  MoveL (T6208) to (121.16, 117.66, 7.9) mm, rotated rx 180 ry 0 rz -180 deg; joints [0, 0, 0, 0, 0, 0]
  Call Extruder 0.15054
  MoveL (T6209) to (117.66, 121.16, 7.9) mm, rotated rx 180 ry 0 rz -180 deg; joints [0, 0, 0, 0, 0, 0]
  Call Extruder 0.03385
  MoveL (T6210) to (116.55, 121.16, 7.9) mm, rotated rx 180 ry 0 rz -180 deg; joints [0, 0, 0, 0, 0, 0]
  Call Extruder 0.54738
  MoveL (T6211) to (103.84, 108.45, 7.9) mm, rotated rx 180 ry 0 rz -180 deg; joints [0, 0, 0, 0, 0, 0]
  Call Extruder 0.03385
  MoveL (T6212) to (103.84, 107.34, 7.9) mm, rotated rx 180 ry 0 rz -180 deg; joints [0, 0, 0, 0, 0, 0]
  Call Extruder 0.15054
  MoveL (T6213) to (107.34, 103.84, 7.9) mm, rotated rx 180 ry 0 rz -180 deg; joints [0, 0, 0, 0, 0, 0]
  Call Extruder 0.10645
  MoveL (T6214) to (103.84, 103.84, 7.9) mm, rotated rx 180 ry 0 rz -180 deg; joints [0, 0, 0, 0, 0, 0]
  Call Extruder 0.7458
  MoveL (T6215) to (121.16, 121.16, 7.9) mm, rotated rx 180 ry 0 rz -180 deg; joints [0, 0, 0, 0, 0, 0]
  Call Extruder 0.07441
  MoveL (T6216) to (118.71, 121.16, 7.9) mm, rotated rx 180 ry 0 rz -180 deg; joints [0, 0, 0, 0, 0, 0]
  Set speed (45.0 mm/s)
  Call Extruder -1.6
  MoveL (T6217) to (118.71, 121.16, 7.9) mm, rotated rx 180 ry 0 rz -180 deg; joints [0, 0, 0, 0, 0, 0]
  Set speed (120.0 mm/s)
  MoveL (T6218) to (118.71, 121.16, 7.9) mm, rotated rx 180 ry 0 rz -180 deg; joints [0, 0, 0, 0, 0, 0]
  Call Extruder -0.38
  MoveL (T6219) to (119.78, 121.16, 7.9) mm, rotated rx 180 ry 0 rz -180 deg; joints [0, 0, 0, 0, 0, 0]
  Set speed (45.0 mm/s)
  Call Extruder -0.02
  MoveL (T6220) to (119.78, 121.16, 7.9) mm, rotated rx 180 ry 0 rz -180 deg; joints [0, 0, 0, 0, 0, 0]
  Set speed (150.0 mm/s)
  MoveL (T6221) to (119.78, 121.16, 9.9) mm, rotated rx 180 ry 0 rz -180 deg; joints [0, 0, 0, 0, 0, 0]
  MoveL (T6222) to (104.34, 103.54, 9.9) mm, rotated rx 180 ry 0 rz -180 deg; joints [0, 0, 0, 0, 0, 0]
  MoveL (T6223) to (104.34, 103.54, 8.1) mm, rotated rx 180 ry 0 rz -180 deg; joints [0, 0, 0, 0, 0, 0]
  Set speed (40.0 mm/s)
  Call Extruder 2.0
  MoveL (T6224) to (104.34, 103.54, 8.1) mm, rotated rx 180 ry 0 rz -180 deg; joints [0, 0, 0, 0, 0, 0]
  Set speed (25.1 mm/s)
  MoveL (T6225) to (104.34, 103.54, 8.1) mm, rotated rx 180 ry 0 rz -180 deg; joints [0, 0, 0, 0, 0, 0]
  Call Extruder 0.13892
  MoveL (T6226) to (108.9, 103.54, 8.1) mm, rotated rx 180 ry 0 rz -180 deg; joints [0, 0, 0, 0, 0, 0]
  Call Extruder 0.05773
  MoveL (T6227) to (108.9, 105.43, 8.1) mm, rotated rx 180 ry 0 rz -180 deg; joints [0, 0, 0, 0, 0, 0]
  Call Extruder 0.18959
  MoveL (T6228) to (115.12, 105.43, 8.1) mm, rotated rx 180 ry 0 rz -180 deg; joints [0, 0, 0, 0, 0, 0]
  Call Extruder 0.05773
  MoveL (T6229) to (115.12, 103.54, 8.1) mm, rotated rx 180 ry 0 rz -180 deg; joints [0, 0, 0, 0, 0, 0]
  Call Extruder 0.19303
  MoveL (T6230) to (121.46, 103.54, 8.1) mm, rotated rx 180 ry 0 rz -180 deg; joints [0, 0, 0, 0, 0, 0]
  Call Extruder 0.20425
  MoveL (T6231) to (121.46, 110.24, 8.1) mm, rotated rx 180 ry 0 rz -180 deg; joints [0, 0, 0, 0, 0, 0]
  Call Extruder 0.05905
  MoveL (T6232) to (119.52, 110.24, 8.1) mm, rotated rx 180 ry 0 rz -180 deg; joints [0, 0, 0, 0, 0, 0]
  Call Extruder 0.11452
  MoveL (T6233) to (119.52, 114, 8.1) mm, rotated rx 180 ry 0 rz -180 deg; joints [0, 0, 0, 0, 0, 0]
  Call Extruder 0.0591
  MoveL (T6234) to (121.46, 114, 8.1) mm, rotated rx 180 ry 0 rz -180 deg; joints [0, 0, 0, 0, 0, 0]
  Call Extruder 0.2272
  MoveL (T6235) to (121.46, 121.46, 8.1) mm, rotated rx 180 ry 0 rz -180 deg; joints [0, 0, 0, 0, 0, 0]
  Call Extruder 0.54596
  MoveL (T6236) to (103.54, 121.46, 8.1) mm, rotated rx 180 ry 0 rz -180 deg; joints [0, 0, 0, 0, 0, 0]
  Call Extruder 0.54596
  MoveL (T6237) to (103.54, 103.54, 8.1) mm, rotated rx 180 ry 0 rz -180 deg; joints [0, 0, 0, 0, 0, 0]
  Call Extruder 0.02254
  MoveL (T6238) to (104.28, 103.54, 8.1) mm, rotated rx 180 ry 0 rz -180 deg; joints [0, 0, 0, 0, 0, 0]
  Set speed (150.0 mm/s)
  MoveL (T6239) to (103.53, 103.13, 8.1) mm, rotated rx 180 ry 0 rz -180 deg; joints [0, 0, 0, 0, 0, 0]
  Set speed (25.1 mm/s)
  MoveL (T6240) to (103.53, 103.13, 8.1) mm, rotated rx 180 ry 0 rz -180 deg; joints [0, 0, 0, 0, 0, 0]
  Call Extruder 0.1759
  MoveL (T6241) to (109.31, 103.13, 8.1) mm, rotated rx 180 ry 0 rz -180 deg; joints [0, 0, 0, 0, 0, 0]
  Call Extruder 0.05773
  MoveL (T6242) to (109.31, 105.03, 8.1) mm, rotated rx 180 ry 0 rz -180 deg; joints [0, 0, 0, 0, 0, 0]
  Call Extruder 0.1648
  MoveL (T6243) to (114.72, 105.03, 8.1) mm, rotated rx 180 ry 0 rz -180 deg; joints [0, 0, 0, 0, 0, 0]
  Call Extruder 0.05773
  MoveL (T6244) to (114.72, 103.13, 8.1) mm, rotated rx 180 ry 0 rz -180 deg; joints [0, 0, 0, 0, 0, 0]
  Call Extruder 0.21783
  MoveL (T6245) to (121.87, 103.13, 8.1) mm, rotated rx 180 ry 0 rz -180 deg; joints [0, 0, 0, 0, 0, 0]
  Call Extruder 0.22906
  MoveL (T6246) to (121.87, 110.65, 8.1) mm, rotated rx 180 ry 0 rz -180 deg; joints [0, 0, 0, 0, 0, 0]
  Call Extruder 0.05906
  MoveL (T6247) to (119.93, 110.65, 8.1) mm, rotated rx 180 ry 0 rz -180 deg; joints [0, 0, 0, 0, 0, 0]
  Call Extruder 0.08971
  MoveL (T6248) to (119.93, 113.59, 8.1) mm, rotated rx 180 ry 0 rz -180 deg; joints [0, 0, 0, 0, 0, 0]
  Call Extruder 0.0591
  MoveL (T6249) to (121.87, 113.6, 8.1) mm, rotated rx 180 ry 0 rz -180 deg; joints [0, 0, 0, 0, 0, 0]
  Call Extruder 0.25199
  MoveL (T6250) to (121.87, 121.87, 8.1) mm, rotated rx 180 ry 0 rz -180 deg; joints [0, 0, 0, 0, 0, 0]
  Call Extruder 0.57077
  MoveL (T6251) to (103.13, 121.87, 8.1) mm, rotated rx 180 ry 0 rz -180 deg; joints [0, 0, 0, 0, 0, 0]
  Call Extruder 0.57077
  MoveL (T6252) to (103.13, 103.13, 8.1) mm, rotated rx 180 ry 0 rz -180 deg; joints [0, 0, 0, 0, 0, 0]
  Call Extruder 0.01036
  MoveL (T6253) to (103.47, 103.13, 8.1) mm, rotated rx 180 ry 0 rz -180 deg; joints [0, 0, 0, 0, 0, 0]
  Set speed (150.0 mm/s)
  MoveL (T6254) to (102.72, 102.81, 8.1) mm, rotated rx 180 ry 0 rz -180 deg; joints [0, 0, 0, 0, 0, 0]
  Set speed (25.0 mm/s)
  MoveL (T6255) to (102.72, 102.81, 8.1) mm, rotated rx 180 ry 0 rz -180 deg; joints [0, 0, 0, 0, 0, 0]
  Call Extruder 0.00259
  MoveL (T6256) to (102.72, 102.72, 8.1) mm, rotated rx 180 ry 0 rz -180 deg; joints [0, 0, 0, 0, 0, 0]
  Call Extruder 0.21288
  MoveL (T6257) to (109.71, 102.72, 8.1) mm, rotated rx 180 ry 0 rz -180 deg; joints [0, 0, 0, 0, 0, 0]
  Call Extruder 0.05773
  MoveL (T6258) to (109.71, 104.62, 8.1) mm, rotated rx 180 ry 0 rz -180 deg; joints [0, 0, 0, 0, 0, 0]
  Call Extruder 0.06775
  MoveL (T6259) to (111.94, 104.62, 8.1) mm, rotated rx 180 ry 0 rz -180 deg; joints [0, 0, 0, 0, 0, 0]
  Call Extruder 0.05773
  MoveL (T6260) to (111.94, 102.72, 8.1) mm, rotated rx 180 ry 0 rz -180 deg; joints [0, 0, 0, 0, 0, 0]
  Call Extruder 0.00738
  MoveL (T6261) to (112.18, 102.72, 8.1) mm, rotated rx 180 ry 0 rz -180 deg; joints [0, 0, 0, 0, 0, 0]
  Call Extruder 0.05773
  MoveL (T6262) to (112.18, 104.62, 8.1) mm, rotated rx 180 ry 0 rz -180 deg; joints [0, 0, 0, 0, 0, 0]
  Call Extruder 0.06494
  MoveL (T6263) to (114.31, 104.62, 8.1) mm, rotated rx 180 ry 0 rz -180 deg; joints [0, 0, 0, 0, 0, 0]
  Call Extruder 0.05773
  MoveL (T6264) to (114.31, 102.72, 8.1) mm, rotated rx 180 ry 0 rz -180 deg; joints [0, 0, 0, 0, 0, 0]
  Call Extruder 0.24262
  MoveL (T6265) to (122.28, 102.72, 8.1) mm, rotated rx 180 ry 0 rz -180 deg; joints [0, 0, 0, 0, 0, 0]
  Call Extruder 0.25387
  MoveL (T6266) to (122.28, 111.06, 8.1) mm, rotated rx 180 ry 0 rz -180 deg; joints [0, 0, 0, 0, 0, 0]
  Call Extruder 0.05906
  MoveL (T6267) to (120.34, 111.06, 8.1) mm, rotated rx 180 ry 0 rz -180 deg; joints [0, 0, 0, 0, 0, 0]
  Call Extruder 0.06491
  MoveL (T6268) to (120.33, 113.19, 8.1) mm, rotated rx 180 ry 0 rz -180 deg; joints [0, 0, 0, 0, 0, 0]
  Call Extruder 0.05909
  MoveL (T6269) to (122.28, 113.19, 8.1) mm, rotated rx 180 ry 0 rz -180 deg; joints [0, 0, 0, 0, 0, 0]
  Call Extruder 0.27679
  MoveL (T6270) to (122.28, 122.28, 8.1) mm, rotated rx 180 ry 0 rz -180 deg; joints [0, 0, 0, 0, 0, 0]
  Call Extruder 0.59557
  MoveL (T6271) to (102.72, 122.28, 8.1) mm, rotated rx 180 ry 0 rz -180 deg; joints [0, 0, 0, 0, 0, 0]
  Call Extruder 0.59115
  MoveL (T6272) to (102.72, 102.87, 8.1) mm, rotated rx 180 ry 0 rz -180 deg; joints [0, 0, 0, 0, 0, 0]
  Set speed (150.0 mm/s)
  MoveL (T6273) to (102.78, 102.75, 8.1) mm, rotated rx 180 ry 0 rz -180 deg; joints [0, 0, 0, 0, 0, 0]
  Set speed (45.0 mm/s)
  Call Extruder -1.6
  MoveL (T6274) to (102.78, 102.75, 8.1) mm, rotated rx 180 ry 0 rz -180 deg; joints [0, 0, 0, 0, 0, 0]
  Set speed (120.0 mm/s)
  MoveL (T6275) to (102.78, 102.75, 8.1) mm, rotated rx 180 ry 0 rz -180 deg; joints [0, 0, 0, 0, 0, 0]
  Call Extruder -0.05166
  MoveL (T6276) to (102.72, 102.72, 8.1) mm, rotated rx 180 ry 0 rz -180 deg; joints [0, 0, 0, 0, 0, 0]
  Call Extruder -0.32834
  MoveL (T6277) to (103.65, 102.72, 8.1) mm, rotated rx 180 ry 0 rz -180 deg; joints [0, 0, 0, 0, 0, 0]
  Set speed (45.0 mm/s)
  Call Extruder -0.02
  MoveL (T6278) to (103.65, 102.72, 8.1) mm, rotated rx 180 ry 0 rz -180 deg; joints [0, 0, 0, 0, 0, 0]
  Set speed (150.0 mm/s)
  MoveL (T6279) to (103.65, 102.72, 10.1) mm, rotated rx 180 ry 0 rz -180 deg; joints [0, 0, 0, 0, 0, 0]
  MoveL (T6280) to (108.78, 104.69, 10.1) mm, rotated rx 180 ry 0 rz -180 deg; joints [0, 0, 0, 0, 0, 0]
  MoveL (T6281) to (108.78, 104.69, 8.1) mm, rotated rx 180 ry 0 rz -180 deg; joints [0, 0, 0, 0, 0, 0]
  Set speed (40.0 mm/s)
  Call Extruder 2.0
  MoveL (T6282) to (108.78, 104.69, 8.1) mm, rotated rx 180 ry 0 rz -180 deg; joints [0, 0, 0, 0, 0, 0]
  Set speed (25.1 mm/s)
  MoveL (T6283) to (108.78, 104.69, 8.1) mm, rotated rx 180 ry 0 rz -180 deg; joints [0, 0, 0, 0, 0, 0]
  Call Extruder 0.01598
  MoveL (T6284) to (108.43, 105.04, 8.1) mm, rotated rx 180 ry 0 rz -180 deg; joints [0, 0, 0, 0, 0, 0]
  Call Extruder 0.01987
  MoveL (T6285) to (108.43, 104.43, 8.1) mm, rotated rx 180 ry 0 rz -180 deg; joints [0, 0, 0, 0, 0, 0]
  Call Extruder 0.01598
  MoveL (T6286) to (108.78, 104.08, 8.1) mm, rotated rx 180 ry 0 rz -180 deg; joints [0, 0, 0, 0, 0, 0]
  Set speed (45.0 mm/s)
  Call Extruder -1.6
  MoveL (T6287) to (108.78, 104.08, 8.1) mm, rotated rx 180 ry 0 rz -180 deg; joints [0, 0, 0, 0, 0, 0]
  Set speed (120.0 mm/s)
  MoveL (T6288) to (108.78, 104.08, 8.1) mm, rotated rx 180 ry 0 rz -180 deg; joints [0, 0, 0, 0, 0, 0]
  Call Extruder -0.17547
  MoveL (T6289) to (108.43, 104.43, 8.1) mm, rotated rx 180 ry 0 rz -180 deg; joints [0, 0, 0, 0, 0, 0]
  Call Extruder -0.20453
  MoveL (T6290) to (108.43, 105, 8.1) mm, rotated rx 180 ry 0 rz -180 deg; joints [0, 0, 0, 0, 0, 0]
  Set speed (45.0 mm/s)
  Call Extruder -0.02
  MoveL (T6291) to (108.43, 105, 8.1) mm, rotated rx 180 ry 0 rz -180 deg; joints [0, 0, 0, 0, 0, 0]
  Set speed (150.0 mm/s)
  MoveL (T6292) to (108.43, 105, 10.1) mm, rotated rx 180 ry 0 rz -180 deg; joints [0, 0, 0, 0, 0, 0]
  MoveL (T6293) to (115.13, 105.79, 10.1) mm, rotated rx 180 ry 0 rz -180 deg; joints [0, 0, 0, 0, 0, 0]
  MoveL (T6294) to (115.13, 105.79, 8.1) mm, rotated rx 180 ry 0 rz -180 deg; joints [0, 0, 0, 0, 0, 0]
  Set speed (40.0 mm/s)
  Call Extruder 2.0
  MoveL (T6295) to (115.13, 105.79, 8.1) mm, rotated rx 180 ry 0 rz -180 deg; joints [0, 0, 0, 0, 0, 0]
  Set speed (25.1 mm/s)
  MoveL (T6296) to (115.13, 105.79, 8.1) mm, rotated rx 180 ry 0 rz -180 deg; joints [0, 0, 0, 0, 0, 0]
  Call Extruder 0.00342
  MoveL (T6297) to (115.21, 105.87, 8.1) mm, rotated rx 180 ry 0 rz -180 deg; joints [0, 0, 0, 0, 0, 0]
  Call Extruder 0.01615
  MoveL (T6298) to (115.74, 105.87, 8.1) mm, rotated rx 180 ry 0 rz -180 deg; joints [0, 0, 0, 0, 0, 0]
  Call Extruder 0.01375
  MoveL (T6299) to (116.06, 105.55, 8.1) mm, rotated rx 180 ry 0 rz -180 deg; joints [0, 0, 0, 0, 0, 0]
  Call Extruder 0.03706
  MoveL (T6300) to (116.06, 104.33, 8.1) mm, rotated rx 180 ry 0 rz -180 deg; joints [0, 0, 0, 0, 0, 0]
  Call Extruder 0.02096
  MoveL (T6301) to (116.55, 103.84, 8.1) mm, rotated rx 180 ry 0 rz -180 deg; joints [0, 0, 0, 0, 0, 0]
  Call Extruder 0.03385
  MoveL (T6302) to (117.66, 103.84, 8.1) mm, rotated rx 180 ry 0 rz -180 deg; joints [0, 0, 0, 0, 0, 0]
  Call Extruder 0.15054
  MoveL (T6303) to (121.16, 107.34, 8.1) mm, rotated rx 180 ry 0 rz -180 deg; joints [0, 0, 0, 0, 0, 0]
  Call Extruder 0.03385
  MoveL (T6304) to (121.16, 108.45, 8.1) mm, rotated rx 180 ry 0 rz -180 deg; joints [0, 0, 0, 0, 0, 0]
  Call Extruder 0.06409
  MoveL (T6305) to (119.67, 109.94, 8.1) mm, rotated rx 180 ry 0 rz -180 deg; joints [0, 0, 0, 0, 0, 0]
  Call Extruder 0.04532
  MoveL (T6306) to (121.16, 109.94, 8.1) mm, rotated rx 180 ry 0 rz -180 deg; joints [0, 0, 0, 0, 0, 0]
  Call Extruder 0.02909
  MoveL (T6307) to (121.16, 108.98, 8.1) mm, rotated rx 180 ry 0 rz -180 deg; joints [0, 0, 0, 0, 0, 0]
  Set speed (45.0 mm/s)
  Call Extruder -1.6
  MoveL (T6308) to (121.16, 108.98, 8.1) mm, rotated rx 180 ry 0 rz -180 deg; joints [0, 0, 0, 0, 0, 0]
  Set speed (120.0 mm/s)
  MoveL (T6309) to (121.16, 108.98, 8.1) mm, rotated rx 180 ry 0 rz -180 deg; joints [0, 0, 0, 0, 0, 0]
  Call Extruder -0.34013
  MoveL (T6310) to (121.16, 109.94, 8.1) mm, rotated rx 180 ry 0 rz -180 deg; joints [0, 0, 0, 0, 0, 0]
  Call Extruder -0.03987
  MoveL (T6311) to (121.04, 109.94, 8.1) mm, rotated rx 180 ry 0 rz -180 deg; joints [0, 0, 0, 0, 0, 0]
  Set speed (45.0 mm/s)
  Call Extruder -0.02
  MoveL (T6312) to (121.04, 109.94, 8.1) mm, rotated rx 180 ry 0 rz -180 deg; joints [0, 0, 0, 0, 0, 0]
  Set speed (150.0 mm/s)
  MoveL (T6313) to (121.04, 109.94, 10.1) mm, rotated rx 180 ry 0 rz -180 deg; joints [0, 0, 0, 0, 0, 0]
  MoveL (T6314) to (118.71, 103.84, 10.1) mm, rotated rx 180 ry 0 rz -180 deg; joints [0, 0, 0, 0, 0, 0]
  MoveL (T6315) to (118.71, 103.84, 8.1) mm, rotated rx 180 ry 0 rz -180 deg; joints [0, 0, 0, 0, 0, 0]
  Set speed (40.0 mm/s)
  Call Extruder 2.0
  MoveL (T6316) to (118.71, 103.84, 8.1) mm, rotated rx 180 ry 0 rz -180 deg; joints [0, 0, 0, 0, 0, 0]
  Set speed (25.1 mm/s)
  MoveL (T6317) to (118.71, 103.84, 8.1) mm, rotated rx 180 ry 0 rz -180 deg; joints [0, 0, 0, 0, 0, 0]
  Call Extruder 0.07441
  MoveL (T6318) to (121.16, 103.84, 8.1) mm, rotated rx 180 ry 0 rz -180 deg; joints [0, 0, 0, 0, 0, 0]
  Call Extruder 0.7458
  MoveL (T6319) to (103.84, 121.16, 8.1) mm, rotated rx 180 ry 0 rz -180 deg; joints [0, 0, 0, 0, 0, 0]
  Call Extruder 0.10645
  MoveL (T6320) to (103.84, 117.66, 8.1) mm, rotated rx 180 ry 0 rz -180 deg; joints [0, 0, 0, 0, 0, 0]
  Call Extruder 0.15054
  MoveL (T6321) to (107.34, 121.16, 8.1) mm, rotated rx 180 ry 0 rz -180 deg; joints [0, 0, 0, 0, 0, 0]
  Call Extruder 0.03385
  MoveL (T6322) to (108.45, 121.16, 8.1) mm, rotated rx 180 ry 0 rz -180 deg; joints [0, 0, 0, 0, 0, 0]
  Call Extruder 0.46387
  MoveL (T6323) to (119.22, 110.39, 8.1) mm, rotated rx 180 ry 0 rz -180 deg; joints [0, 0, 0, 0, 0, 0]
  Call Extruder 0.01165
  MoveL (T6324) to (119.22, 110.01, 8.1) mm, rotated rx 180 ry 0 rz -180 deg; joints [0, 0, 0, 0, 0, 0]
  Call Extruder 0.18382
  MoveL (T6325) to (114.95, 105.74, 8.1) mm, rotated rx 180 ry 0 rz -180 deg; joints [0, 0, 0, 0, 0, 0]
  Call Extruder 0.009
  MoveL (T6326) to (114.66, 105.74, 8.1) mm, rotated rx 180 ry 0 rz -180 deg; joints [0, 0, 0, 0, 0, 0]
  Call Extruder 0.46575
  MoveL (T6327) to (103.84, 116.55, 8.1) mm, rotated rx 180 ry 0 rz -180 deg; joints [0, 0, 0, 0, 0, 0]
  Call Extruder 0.07441
  MoveL (T6328) to (103.84, 114.11, 8.1) mm, rotated rx 180 ry 0 rz -180 deg; joints [0, 0, 0, 0, 0, 0]
  Set speed (45.0 mm/s)
  Call Extruder -1.6
  MoveL (T6329) to (103.84, 114.11, 8.1) mm, rotated rx 180 ry 0 rz -180 deg; joints [0, 0, 0, 0, 0, 0]
  Set speed (120.0 mm/s)
  MoveL (T6330) to (103.84, 114.11, 8.1) mm, rotated rx 180 ry 0 rz -180 deg; joints [0, 0, 0, 0, 0, 0]
  Call Extruder -0.38
  MoveL (T6331) to (103.84, 115.17, 8.1) mm, rotated rx 180 ry 0 rz -180 deg; joints [0, 0, 0, 0, 0, 0]
  Set speed (45.0 mm/s)
  Call Extruder -0.02
  MoveL (T6332) to (103.84, 115.17, 8.1) mm, rotated rx 180 ry 0 rz -180 deg; joints [0, 0, 0, 0, 0, 0]
  Set speed (150.0 mm/s)
  MoveL (T6333) to (103.84, 115.17, 10.1) mm, rotated rx 180 ry 0 rz -180 deg; joints [0, 0, 0, 0, 0, 0]
  MoveL (T6334) to (115.37, 105.64, 10.1) mm, rotated rx 180 ry 0 rz -180 deg; joints [0, 0, 0, 0, 0, 0]
  MoveL (T6335) to (115.37, 105.64, 8.1) mm, rotated rx 180 ry 0 rz -180 deg; joints [0, 0, 0, 0, 0, 0]
  Set speed (40.0 mm/s)
  Call Extruder 2.0
  MoveL (T6336) to (115.37, 105.64, 8.1) mm, rotated rx 180 ry 0 rz -180 deg; joints [0, 0, 0, 0, 0, 0]
  Set speed (25.1 mm/s)
  MoveL (T6337) to (115.37, 105.64, 8.1) mm, rotated rx 180 ry 0 rz -180 deg; joints [0, 0, 0, 0, 0, 0]
  Call Extruder 0.01303
  MoveL (T6338) to (115.66, 105.36, 8.1) mm, rotated rx 180 ry 0 rz -180 deg; joints [0, 0, 0, 0, 0, 0]
  Call Extruder 0.01995
  MoveL (T6339) to (115.66, 104.75, 8.1) mm, rotated rx 180 ry 0 rz -180 deg; joints [0, 0, 0, 0, 0, 0]
  Call Extruder 0.01043
  MoveL (T6340) to (115.43, 104.97, 8.1) mm, rotated rx 180 ry 0 rz -180 deg; joints [0, 0, 0, 0, 0, 0]
  Call Extruder 0.01995
  MoveL (T6341) to (115.43, 104.36, 8.1) mm, rotated rx 180 ry 0 rz -180 deg; joints [0, 0, 0, 0, 0, 0]
  Call Extruder 0.01885
  MoveL (T6342) to (115.84, 103.95, 8.1) mm, rotated rx 180 ry 0 rz -180 deg; joints [0, 0, 0, 0, 0, 0]
  Set speed (45.0 mm/s)
  Call Extruder -1.6
  MoveL (T6343) to (115.84, 103.95, 8.1) mm, rotated rx 180 ry 0 rz -180 deg; joints [0, 0, 0, 0, 0, 0]
  Set speed (120.0 mm/s)
  MoveL (T6344) to (115.84, 103.95, 8.1) mm, rotated rx 180 ry 0 rz -180 deg; joints [0, 0, 0, 0, 0, 0]
  Call Extruder -0.20676
  MoveL (T6345) to (115.43, 104.36, 8.1) mm, rotated rx 180 ry 0 rz -180 deg; joints [0, 0, 0, 0, 0, 0]
  Call Extruder -0.17324
  MoveL (T6346) to (115.43, 104.84, 8.1) mm, rotated rx 180 ry 0 rz -180 deg; joints [0, 0, 0, 0, 0, 0]
  Set speed (45.0 mm/s)
  Call Extruder -0.02
  MoveL (T6347) to (115.43, 104.84, 8.1) mm, rotated rx 180 ry 0 rz -180 deg; joints [0, 0, 0, 0, 0, 0]
  Set speed (150.0 mm/s)
  MoveL (T6348) to (115.43, 104.84, 10.1) mm, rotated rx 180 ry 0 rz -180 deg; joints [0, 0, 0, 0, 0, 0]
  MoveL (T6349) to (121.16, 115.5, 10.1) mm, rotated rx 180 ry 0 rz -180 deg; joints [0, 0, 0, 0, 0, 0]
  MoveL (T6350) to (121.16, 115.5, 8.1) mm, rotated rx 180 ry 0 rz -180 deg; joints [0, 0, 0, 0, 0, 0]
  Set speed (40.0 mm/s)
  Call Extruder 2.0
  MoveL (T6351) to (121.16, 115.5, 8.1) mm, rotated rx 180 ry 0 rz -180 deg; joints [0, 0, 0, 0, 0, 0]
  Set speed (25.1 mm/s)
  MoveL (T6352) to (121.16, 115.5, 8.1) mm, rotated rx 180 ry 0 rz -180 deg; joints [0, 0, 0, 0, 0, 0]
  Call Extruder 0.03627
  MoveL (T6353) to (121.16, 114.31, 8.1) mm, rotated rx 180 ry 0 rz -180 deg; joints [0, 0, 0, 0, 0, 0]
  Call Extruder 0.03814
  MoveL (T6354) to (119.9, 114.31, 8.1) mm, rotated rx 180 ry 0 rz -180 deg; joints [0, 0, 0, 0, 0, 0]
  Call Extruder 0.29503
  MoveL (T6355) to (113.06, 121.16, 8.1) mm, rotated rx 180 ry 0 rz -180 deg; joints [0, 0, 0, 0, 0, 0]
  Call Extruder 0.03385
  MoveL (T6356) to (111.94, 121.16, 8.1) mm, rotated rx 180 ry 0 rz -180 deg; joints [0, 0, 0, 0, 0, 0]
  Call Extruder 0.34896
  MoveL (T6357) to (103.84, 113.06, 8.1) mm, rotated rx 180 ry 0 rz -180 deg; joints [0, 0, 0, 0, 0, 0]
  Call Extruder 0.03385
  MoveL (T6358) to (103.84, 111.94, 8.1) mm, rotated rx 180 ry 0 rz -180 deg; joints [0, 0, 0, 0, 0, 0]
  Call Extruder 0.26733
  MoveL (T6359) to (110.05, 105.74, 8.1) mm, rotated rx 180 ry 0 rz -180 deg; joints [0, 0, 0, 0, 0, 0]
  Call Extruder 0.009
  MoveL (T6360) to (110.34, 105.74, 8.1) mm, rotated rx 180 ry 0 rz -180 deg; joints [0, 0, 0, 0, 0, 0]
  Call Extruder 0.46575
  MoveL (T6361) to (121.16, 116.55, 8.1) mm, rotated rx 180 ry 0 rz -180 deg; joints [0, 0, 0, 0, 0, 0]
  Call Extruder 0.03385
  MoveL (T6362) to (121.16, 117.66, 8.1) mm, rotated rx 180 ry 0 rz -180 deg; joints [0, 0, 0, 0, 0, 0]
  Call Extruder 0.15054
  MoveL (T6363) to (117.66, 121.16, 8.1) mm, rotated rx 180 ry 0 rz -180 deg; joints [0, 0, 0, 0, 0, 0]
  Call Extruder 0.03385
  MoveL (T6364) to (116.55, 121.16, 8.1) mm, rotated rx 180 ry 0 rz -180 deg; joints [0, 0, 0, 0, 0, 0]
  Call Extruder 0.54738
  MoveL (T6365) to (103.84, 108.45, 8.1) mm, rotated rx 180 ry 0 rz -180 deg; joints [0, 0, 0, 0, 0, 0]
  Call Extruder 0.03385
  MoveL (T6366) to (103.84, 107.34, 8.1) mm, rotated rx 180 ry 0 rz -180 deg; joints [0, 0, 0, 0, 0, 0]
  Call Extruder 0.15054
  MoveL (T6367) to (107.34, 103.84, 8.1) mm, rotated rx 180 ry 0 rz -180 deg; joints [0, 0, 0, 0, 0, 0]
  Call Extruder 0.10645
  MoveL (T6368) to (103.84, 103.84, 8.1) mm, rotated rx 180 ry 0 rz -180 deg; joints [0, 0, 0, 0, 0, 0]
  Call Extruder 0.7458
  MoveL (T6369) to (121.16, 121.16, 8.1) mm, rotated rx 180 ry 0 rz -180 deg; joints [0, 0, 0, 0, 0, 0]
  Call Extruder 0.07441
  MoveL (T6370) to (118.71, 121.16, 8.1) mm, rotated rx 180 ry 0 rz -180 deg; joints [0, 0, 0, 0, 0, 0]
  Set speed (45.0 mm/s)
  Call Extruder -1.6
  MoveL (T6371) to (118.71, 121.16, 8.1) mm, rotated rx 180 ry 0 rz -180 deg; joints [0, 0, 0, 0, 0, 0]
  Set speed (120.0 mm/s)
  MoveL (T6372) to (118.71, 121.16, 8.1) mm, rotated rx 180 ry 0 rz -180 deg; joints [0, 0, 0, 0, 0, 0]
  Call Extruder -0.38
  MoveL (T6373) to (119.78, 121.16, 8.1) mm, rotated rx 180 ry 0 rz -180 deg; joints [0, 0, 0, 0, 0, 0]
  Set speed (45.0 mm/s)
  Call Extruder -0.02
  MoveL (T6374) to (119.78, 121.16, 8.1) mm, rotated rx 180 ry 0 rz -180 deg; joints [0, 0, 0, 0, 0, 0]
  Set speed (150.0 mm/s)
  MoveL (T6375) to (119.78, 121.16, 10.1) mm, rotated rx 180 ry 0 rz -180 deg; joints [0, 0, 0, 0, 0, 0]
  MoveL (T6376) to (112.06, 102.81, 10.1) mm, rotated rx 180 ry 0 rz -180 deg; joints [0, 0, 0, 0, 0, 0]
  MoveL (T6377) to (112.06, 102.81, 8.3) mm, rotated rx 180 ry 0 rz -180 deg; joints [0, 0, 0, 0, 0, 0]
  Set speed (40.0 mm/s)
  Call Extruder 2.0
  MoveL (T6378) to (112.06, 102.81, 8.3) mm, rotated rx 180 ry 0 rz -180 deg; joints [0, 0, 0, 0, 0, 0]
  Set speed (25.0 mm/s)
  MoveL (T6379) to (112.06, 102.81, 8.3) mm, rotated rx 180 ry 0 rz -180 deg; joints [0, 0, 0, 0, 0, 0]
  Call Extruder 0.00245
  MoveL (T6380) to (112.06, 102.72, 8.3) mm, rotated rx 180 ry 0 rz -180 deg; joints [0, 0, 0, 0, 0, 0]
  Call Extruder 0.05685
  MoveL (T6381) to (112.06, 104.59, 8.3) mm, rotated rx 180 ry 0 rz -180 deg; joints [0, 0, 0, 0, 0, 0]
  Call Extruder 0.05257
  MoveL (T6382) to (112.06, 102.86, 8.3) mm, rotated rx 180 ry 0 rz -180 deg; joints [0, 0, 0, 0, 0, 0]
  Set speed (150.0 mm/s)
  MoveL (T6383) to (112.12, 102.85, 8.3) mm, rotated rx 180 ry 0 rz -180 deg; joints [0, 0, 0, 0, 0, 0]
  Set speed (45.0 mm/s)
  Call Extruder -1.6
  MoveL (T6384) to (112.12, 102.85, 8.3) mm, rotated rx 180 ry 0 rz -180 deg; joints [0, 0, 0, 0, 0, 0]
  Set speed (120.0 mm/s)
  MoveL (T6385) to (112.12, 102.85, 8.3) mm, rotated rx 180 ry 0 rz -180 deg; joints [0, 0, 0, 0, 0, 0]
  Call Extruder -0.05002
  MoveL (T6386) to (112.06, 102.72, 8.3) mm, rotated rx 180 ry 0 rz -180 deg; joints [0, 0, 0, 0, 0, 0]
  Call Extruder -0.32998
  MoveL (T6387) to (112.06, 103.65, 8.3) mm, rotated rx 180 ry 0 rz -180 deg; joints [0, 0, 0, 0, 0, 0]
  Set speed (45.0 mm/s)
  Call Extruder -0.02
  MoveL (T6388) to (112.06, 103.65, 8.3) mm, rotated rx 180 ry 0 rz -180 deg; joints [0, 0, 0, 0, 0, 0]
  Set speed (150.0 mm/s)
  MoveL (T6389) to (112.06, 103.65, 10.3) mm, rotated rx 180 ry 0 rz -180 deg; joints [0, 0, 0, 0, 0, 0]
  MoveL (T6390) to (104.34, 103.54, 10.3) mm, rotated rx 180 ry 0 rz -180 deg; joints [0, 0, 0, 0, 0, 0]
  MoveL (T6391) to (104.34, 103.54, 8.3) mm, rotated rx 180 ry 0 rz -180 deg; joints [0, 0, 0, 0, 0, 0]
  Set speed (40.0 mm/s)
  Call Extruder 2.0
  MoveL (T6392) to (104.34, 103.54, 8.3) mm, rotated rx 180 ry 0 rz -180 deg; joints [0, 0, 0, 0, 0, 0]
  Set speed (25.0 mm/s)
  MoveL (T6393) to (104.34, 103.54, 8.3) mm, rotated rx 180 ry 0 rz -180 deg; joints [0, 0, 0, 0, 0, 0]
  Call Extruder 0.1423
  MoveL (T6394) to (109.01, 103.54, 8.3) mm, rotated rx 180 ry 0 rz -180 deg; joints [0, 0, 0, 0, 0, 0]
  Call Extruder 0.05773
  MoveL (T6395) to (109.01, 105.43, 8.3) mm, rotated rx 180 ry 0 rz -180 deg; joints [0, 0, 0, 0, 0, 0]
  Call Extruder 0.18235
  MoveL (T6396) to (115, 105.43, 8.3) mm, rotated rx 180 ry 0 rz -180 deg; joints [0, 0, 0, 0, 0, 0]
  Call Extruder 0.05773
  MoveL (T6397) to (115, 103.54, 8.3) mm, rotated rx 180 ry 0 rz -180 deg; joints [0, 0, 0, 0, 0, 0]
  Call Extruder 0.19688
  MoveL (T6398) to (121.46, 103.54, 8.3) mm, rotated rx 180 ry 0 rz -180 deg; joints [0, 0, 0, 0, 0, 0]
  Call Extruder 0.20419
  MoveL (T6399) to (121.46, 110.24, 8.3) mm, rotated rx 180 ry 0 rz -180 deg; joints [0, 0, 0, 0, 0, 0]
  Call Extruder 0.05904
  MoveL (T6400) to (119.52, 110.24, 8.3) mm, rotated rx 180 ry 0 rz -180 deg; joints [0, 0, 0, 0, 0, 0]
  Call Extruder 0.11452
  MoveL (T6401) to (119.52, 114, 8.3) mm, rotated rx 180 ry 0 rz -180 deg; joints [0, 0, 0, 0, 0, 0]
  Call Extruder 0.05909
  MoveL (T6402) to (121.46, 114, 8.3) mm, rotated rx 180 ry 0 rz -180 deg; joints [0, 0, 0, 0, 0, 0]
  Call Extruder 0.22726
  MoveL (T6403) to (121.46, 121.46, 8.3) mm, rotated rx 180 ry 0 rz -180 deg; joints [0, 0, 0, 0, 0, 0]
  Call Extruder 0.54596
  MoveL (T6404) to (103.54, 121.46, 8.3) mm, rotated rx 180 ry 0 rz -180 deg; joints [0, 0, 0, 0, 0, 0]
  Call Extruder 0.54596
  MoveL (T6405) to (103.54, 103.54, 8.3) mm, rotated rx 180 ry 0 rz -180 deg; joints [0, 0, 0, 0, 0, 0]
  Call Extruder 0.02254
  MoveL (T6406) to (104.28, 103.54, 8.3) mm, rotated rx 180 ry 0 rz -180 deg; joints [0, 0, 0, 0, 0, 0]
  Set speed (150.0 mm/s)
  MoveL (T6407) to (103.53, 103.13, 8.3) mm, rotated rx 180 ry 0 rz -180 deg; joints [0, 0, 0, 0, 0, 0]
  Set speed (25.0 mm/s)
  MoveL (T6408) to (103.53, 103.13, 8.3) mm, rotated rx 180 ry 0 rz -180 deg; joints [0, 0, 0, 0, 0, 0]
  Call Extruder 0.17928
  MoveL (T6409) to (109.42, 103.13, 8.3) mm, rotated rx 180 ry 0 rz -180 deg; joints [0, 0, 0, 0, 0, 0]
  Call Extruder 0.05773
  MoveL (T6410) to (109.42, 105.03, 8.3) mm, rotated rx 180 ry 0 rz -180 deg; joints [0, 0, 0, 0, 0, 0]
  Call Extruder 0.15756
  MoveL (T6411) to (114.59, 105.03, 8.3) mm, rotated rx 180 ry 0 rz -180 deg; joints [0, 0, 0, 0, 0, 0]
  Call Extruder 0.05773
  MoveL (T6412) to (114.59, 103.13, 8.3) mm, rotated rx 180 ry 0 rz -180 deg; joints [0, 0, 0, 0, 0, 0]
  Call Extruder 0.22168
  MoveL (T6413) to (121.87, 103.13, 8.3) mm, rotated rx 180 ry 0 rz -180 deg; joints [0, 0, 0, 0, 0, 0]
  Call Extruder 0.22899
  MoveL (T6414) to (121.87, 110.65, 8.3) mm, rotated rx 180 ry 0 rz -180 deg; joints [0, 0, 0, 0, 0, 0]
  Call Extruder 0.05905
  MoveL (T6415) to (119.93, 110.65, 8.3) mm, rotated rx 180 ry 0 rz -180 deg; joints [0, 0, 0, 0, 0, 0]
  Call Extruder 0.08971
  MoveL (T6416) to (119.93, 113.59, 8.3) mm, rotated rx 180 ry 0 rz -180 deg; joints [0, 0, 0, 0, 0, 0]
  Call Extruder 0.05909
  MoveL (T6417) to (121.87, 113.59, 8.3) mm, rotated rx 180 ry 0 rz -180 deg; joints [0, 0, 0, 0, 0, 0]
  Call Extruder 0.25206
  MoveL (T6418) to (121.87, 121.87, 8.3) mm, rotated rx 180 ry 0 rz -180 deg; joints [0, 0, 0, 0, 0, 0]
  Call Extruder 0.57077
  MoveL (T6419) to (103.13, 121.87, 8.3) mm, rotated rx 180 ry 0 rz -180 deg; joints [0, 0, 0, 0, 0, 0]
  Call Extruder 0.57077
  MoveL (T6420) to (103.13, 103.13, 8.3) mm, rotated rx 180 ry 0 rz -180 deg; joints [0, 0, 0, 0, 0, 0]
  Call Extruder 0.01036
  MoveL (T6421) to (103.47, 103.13, 8.3) mm, rotated rx 180 ry 0 rz -180 deg; joints [0, 0, 0, 0, 0, 0]
  Set speed (150.0 mm/s)
  MoveL (T6422) to (102.72, 102.81, 8.3) mm, rotated rx 180 ry 0 rz -180 deg; joints [0, 0, 0, 0, 0, 0]
  Set speed (25.0 mm/s)
  MoveL (T6423) to (102.72, 102.81, 8.3) mm, rotated rx 180 ry 0 rz -180 deg; joints [0, 0, 0, 0, 0, 0]
  Call Extruder 0.00259
  MoveL (T6424) to (102.72, 102.72, 8.3) mm, rotated rx 180 ry 0 rz -180 deg; joints [0, 0, 0, 0, 0, 0]
  Call Extruder 0.21626
  MoveL (T6425) to (109.82, 102.72, 8.3) mm, rotated rx 180 ry 0 rz -180 deg; joints [0, 0, 0, 0, 0, 0]
  Call Extruder 0.05773
  MoveL (T6426) to (109.83, 104.62, 8.3) mm, rotated rx 180 ry 0 rz -180 deg; joints [0, 0, 0, 0, 0, 0]
  Call Extruder 0.13277
  MoveL (T6427) to (114.18, 104.62, 8.3) mm, rotated rx 180 ry 0 rz -180 deg; joints [0, 0, 0, 0, 0, 0]
  Call Extruder 0.05773
  MoveL (T6428) to (114.18, 102.72, 8.3) mm, rotated rx 180 ry 0 rz -180 deg; joints [0, 0, 0, 0, 0, 0]
  Call Extruder 0.24647
  MoveL (T6429) to (122.28, 102.72, 8.3) mm, rotated rx 180 ry 0 rz -180 deg; joints [0, 0, 0, 0, 0, 0]
  Call Extruder 0.2538
  MoveL (T6430) to (122.28, 111.06, 8.3) mm, rotated rx 180 ry 0 rz -180 deg; joints [0, 0, 0, 0, 0, 0]
  Call Extruder 0.05905
  MoveL (T6431) to (120.34, 111.06, 8.3) mm, rotated rx 180 ry 0 rz -180 deg; joints [0, 0, 0, 0, 0, 0]
  Call Extruder 0.06491
  MoveL (T6432) to (120.34, 113.19, 8.3) mm, rotated rx 180 ry 0 rz -180 deg; joints [0, 0, 0, 0, 0, 0]
  Call Extruder 0.05908
  MoveL (T6433) to (122.28, 113.19, 8.3) mm, rotated rx 180 ry 0 rz -180 deg; joints [0, 0, 0, 0, 0, 0]
  Call Extruder 0.27686
  MoveL (T6434) to (122.28, 122.28, 8.3) mm, rotated rx 180 ry 0 rz -180 deg; joints [0, 0, 0, 0, 0, 0]
  Call Extruder 0.59557
  MoveL (T6435) to (102.72, 122.28, 8.3) mm, rotated rx 180 ry 0 rz -180 deg; joints [0, 0, 0, 0, 0, 0]
  Call Extruder 0.59115
  MoveL (T6436) to (102.72, 102.87, 8.3) mm, rotated rx 180 ry 0 rz -180 deg; joints [0, 0, 0, 0, 0, 0]
  Set speed (150.0 mm/s)
  MoveL (T6437) to (102.78, 102.75, 8.3) mm, rotated rx 180 ry 0 rz -180 deg; joints [0, 0, 0, 0, 0, 0]
  Set speed (45.0 mm/s)
  Call Extruder -1.6
  MoveL (T6438) to (102.78, 102.75, 8.3) mm, rotated rx 180 ry 0 rz -180 deg; joints [0, 0, 0, 0, 0, 0]
  Set speed (120.0 mm/s)
  MoveL (T6439) to (102.78, 102.75, 8.3) mm, rotated rx 180 ry 0 rz -180 deg; joints [0, 0, 0, 0, 0, 0]
  Call Extruder -0.05166
  MoveL (T6440) to (102.72, 102.72, 8.3) mm, rotated rx 180 ry 0 rz -180 deg; joints [0, 0, 0, 0, 0, 0]
  Call Extruder -0.32834
  MoveL (T6441) to (103.65, 102.72, 8.3) mm, rotated rx 180 ry 0 rz -180 deg; joints [0, 0, 0, 0, 0, 0]
  Set speed (45.0 mm/s)
  Call Extruder -0.02
  MoveL (T6442) to (103.65, 102.72, 8.3) mm, rotated rx 180 ry 0 rz -180 deg; joints [0, 0, 0, 0, 0, 0]
  Set speed (150.0 mm/s)
  MoveL (T6443) to (103.65, 102.72, 10.3) mm, rotated rx 180 ry 0 rz -180 deg; joints [0, 0, 0, 0, 0, 0]
  MoveL (T6444) to (108.36, 103.99, 10.3) mm, rotated rx 180 ry 0 rz -180 deg; joints [0, 0, 0, 0, 0, 0]
  MoveL (T6445) to (108.36, 103.99, 8.3) mm, rotated rx 180 ry 0 rz -180 deg; joints [0, 0, 0, 0, 0, 0]
  Set speed (40.0 mm/s)
  Call Extruder 2.0
  MoveL (T6446) to (108.36, 103.99, 8.3) mm, rotated rx 180 ry 0 rz -180 deg; joints [0, 0, 0, 0, 0, 0]
  Set speed (25.0 mm/s)
  MoveL (T6447) to (108.36, 103.99, 8.3) mm, rotated rx 180 ry 0 rz -180 deg; joints [0, 0, 0, 0, 0, 0]
  Call Extruder 0.01562
  MoveL (T6448) to (108.7, 104.34, 8.3) mm, rotated rx 180 ry 0 rz -180 deg; joints [0, 0, 0, 0, 0, 0]
  Call Extruder 0.01897
  MoveL (T6449) to (108.71, 104.94, 8.3) mm, rotated rx 180 ry 0 rz -180 deg; joints [0, 0, 0, 0, 0, 0]
  Call Extruder 0.00741
  MoveL (T6450) to (108.54, 104.77, 8.3) mm, rotated rx 180 ry 0 rz -180 deg; joints [0, 0, 0, 0, 0, 0]
  Call Extruder 0.01897
  MoveL (T6451) to (108.54, 105.37, 8.3) mm, rotated rx 180 ry 0 rz -180 deg; joints [0, 0, 0, 0, 0, 0]
  Call Extruder 0.01234
  MoveL (T6452) to (108.82, 105.64, 8.3) mm, rotated rx 180 ry 0 rz -180 deg; joints [0, 0, 0, 0, 0, 0]
  Set speed (45.0 mm/s)
  Call Extruder -1.6
  MoveL (T6453) to (108.82, 105.64, 8.3) mm, rotated rx 180 ry 0 rz -180 deg; joints [0, 0, 0, 0, 0, 0]
  Set speed (120.0 mm/s)
  MoveL (T6454) to (108.82, 105.64, 8.3) mm, rotated rx 180 ry 0 rz -180 deg; joints [0, 0, 0, 0, 0, 0]
  Call Extruder -0.13882
  MoveL (T6455) to (108.54, 105.37, 8.3) mm, rotated rx 180 ry 0 rz -180 deg; joints [0, 0, 0, 0, 0, 0]
  Call Extruder -0.21335
  MoveL (T6456) to (108.54, 104.77, 8.3) mm, rotated rx 180 ry 0 rz -180 deg; joints [0, 0, 0, 0, 0, 0]
  Call Extruder -0.02783
  MoveL (T6457) to (108.6, 104.82, 8.3) mm, rotated rx 180 ry 0 rz -180 deg; joints [0, 0, 0, 0, 0, 0]
  Set speed (45.0 mm/s)
  Call Extruder -0.02
  MoveL (T6458) to (108.6, 104.82, 8.3) mm, rotated rx 180 ry 0 rz -180 deg; joints [0, 0, 0, 0, 0, 0]
  Set speed (150.0 mm/s)
  MoveL (T6459) to (108.6, 104.82, 10.3) mm, rotated rx 180 ry 0 rz -180 deg; joints [0, 0, 0, 0, 0, 0]
  MoveL (T6460) to (103.84, 114.11, 10.3) mm, rotated rx 180 ry 0 rz -180 deg; joints [0, 0, 0, 0, 0, 0]
  MoveL (T6461) to (103.84, 114.11, 8.3) mm, rotated rx 180 ry 0 rz -180 deg; joints [0, 0, 0, 0, 0, 0]
  Set speed (40.0 mm/s)
  Call Extruder 2.0
  MoveL (T6462) to (103.84, 114.11, 8.3) mm, rotated rx 180 ry 0 rz -180 deg; joints [0, 0, 0, 0, 0, 0]
  Set speed (25.0 mm/s)
  MoveL (T6463) to (103.84, 114.11, 8.3) mm, rotated rx 180 ry 0 rz -180 deg; joints [0, 0, 0, 0, 0, 0]
  Call Extruder 0.07441
  MoveL (T6464) to (103.84, 116.55, 8.3) mm, rotated rx 180 ry 0 rz -180 deg; joints [0, 0, 0, 0, 0, 0]
  Call Extruder 0.46574
  MoveL (T6465) to (114.66, 105.74, 8.3) mm, rotated rx 180 ry 0 rz -180 deg; joints [0, 0, 0, 0, 0, 0]
  Call Extruder 0.00901
  MoveL (T6466) to (114.95, 105.74, 8.3) mm, rotated rx 180 ry 0 rz -180 deg; joints [0, 0, 0, 0, 0, 0]
  Call Extruder 0.18383
  MoveL (T6467) to (119.22, 110.01, 8.3) mm, rotated rx 180 ry 0 rz -180 deg; joints [0, 0, 0, 0, 0, 0]
  Call Extruder 0.01163
  MoveL (T6468) to (119.22, 110.39, 8.3) mm, rotated rx 180 ry 0 rz -180 deg; joints [0, 0, 0, 0, 0, 0]
  Call Extruder 0.46388
  MoveL (T6469) to (108.45, 121.16, 8.3) mm, rotated rx 180 ry 0 rz -180 deg; joints [0, 0, 0, 0, 0, 0]
  Call Extruder 0.03385
  MoveL (T6470) to (107.34, 121.16, 8.3) mm, rotated rx 180 ry 0 rz -180 deg; joints [0, 0, 0, 0, 0, 0]
  Call Extruder 0.15054
  MoveL (T6471) to (103.84, 117.66, 8.3) mm, rotated rx 180 ry 0 rz -180 deg; joints [0, 0, 0, 0, 0, 0]
  Call Extruder 0.10645
  MoveL (T6472) to (103.84, 121.16, 8.3) mm, rotated rx 180 ry 0 rz -180 deg; joints [0, 0, 0, 0, 0, 0]
  Call Extruder 0.7458
  MoveL (T6473) to (121.16, 103.84, 8.3) mm, rotated rx 180 ry 0 rz -180 deg; joints [0, 0, 0, 0, 0, 0]
  Call Extruder 0.07441
  MoveL (T6474) to (118.71, 103.84, 8.3) mm, rotated rx 180 ry 0 rz -180 deg; joints [0, 0, 0, 0, 0, 0]
  Set speed (45.0 mm/s)
  Call Extruder -1.6
  MoveL (T6475) to (118.71, 103.84, 8.3) mm, rotated rx 180 ry 0 rz -180 deg; joints [0, 0, 0, 0, 0, 0]
  Set speed (120.0 mm/s)
  MoveL (T6476) to (118.71, 103.84, 8.3) mm, rotated rx 180 ry 0 rz -180 deg; joints [0, 0, 0, 0, 0, 0]
  Call Extruder -0.38
  MoveL (T6477) to (119.78, 103.84, 8.3) mm, rotated rx 180 ry 0 rz -180 deg; joints [0, 0, 0, 0, 0, 0]
  Set speed (45.0 mm/s)
  Call Extruder -0.02
  MoveL (T6478) to (119.78, 103.84, 8.3) mm, rotated rx 180 ry 0 rz -180 deg; joints [0, 0, 0, 0, 0, 0]
  Set speed (150.0 mm/s)
  MoveL (T6479) to (119.78, 103.84, 10.3) mm, rotated rx 180 ry 0 rz -180 deg; joints [0, 0, 0, 0, 0, 0]
  MoveL (T6480) to (115.12, 104.04, 10.3) mm, rotated rx 180 ry 0 rz -180 deg; joints [0, 0, 0, 0, 0, 0]
  MoveL (T6481) to (115.12, 104.04, 8.3) mm, rotated rx 180 ry 0 rz -180 deg; joints [0, 0, 0, 0, 0, 0]
  Set speed (40.0 mm/s)
  Call Extruder 2.0
  MoveL (T6482) to (115.12, 104.04, 8.3) mm, rotated rx 180 ry 0 rz -180 deg; joints [0, 0, 0, 0, 0, 0]
  Set speed (25.0 mm/s)
  MoveL (T6483) to (115.12, 104.04, 8.3) mm, rotated rx 180 ry 0 rz -180 deg; joints [0, 0, 0, 0, 0, 0]
  Call Extruder 0.01928
  MoveL (T6484) to (115.53, 104.45, 8.3) mm, rotated rx 180 ry 0 rz -180 deg; joints [0, 0, 0, 0, 0, 0]
  Call Extruder 0.02088
  MoveL (T6485) to (115.53, 105.08, 8.3) mm, rotated rx 180 ry 0 rz -180 deg; joints [0, 0, 0, 0, 0, 0]
  Call Extruder 0.01928
  MoveL (T6486) to (115.12, 104.67, 8.3) mm, rotated rx 180 ry 0 rz -180 deg; joints [0, 0, 0, 0, 0, 0]
  Set speed (150.0 mm/s)
  MoveL (T6487) to (115.1, 105.87, 8.3) mm, rotated rx 180 ry 0 rz -180 deg; joints [0, 0, 0, 0, 0, 0]
  Set speed (25.0 mm/s)
  MoveL (T6488) to (115.1, 105.87, 8.3) mm, rotated rx 180 ry 0 rz -180 deg; joints [0, 0, 0, 0, 0, 0]
  Call Extruder 0.01572
  MoveL (T6489) to (115.62, 105.87, 8.3) mm, rotated rx 180 ry 0 rz -180 deg; joints [0, 0, 0, 0, 0, 0]
  Call Extruder 0.01375
  MoveL (T6490) to (115.94, 105.55, 8.3) mm, rotated rx 180 ry 0 rz -180 deg; joints [0, 0, 0, 0, 0, 0]
  Call Extruder 0.03321
  MoveL (T6491) to (115.94, 104.46, 8.3) mm, rotated rx 180 ry 0 rz -180 deg; joints [0, 0, 0, 0, 0, 0]
  Call Extruder 0.02641
  MoveL (T6492) to (116.55, 103.84, 8.3) mm, rotated rx 180 ry 0 rz -180 deg; joints [0, 0, 0, 0, 0, 0]
  Call Extruder 0.03385
  MoveL (T6493) to (117.66, 103.84, 8.3) mm, rotated rx 180 ry 0 rz -180 deg; joints [0, 0, 0, 0, 0, 0]
  Call Extruder 0.15054
  MoveL (T6494) to (121.16, 107.34, 8.3) mm, rotated rx 180 ry 0 rz -180 deg; joints [0, 0, 0, 0, 0, 0]
  Call Extruder 0.03385
  MoveL (T6495) to (121.16, 108.45, 8.3) mm, rotated rx 180 ry 0 rz -180 deg; joints [0, 0, 0, 0, 0, 0]
  Call Extruder 0.064
  MoveL (T6496) to (119.67, 109.94, 8.3) mm, rotated rx 180 ry 0 rz -180 deg; joints [0, 0, 0, 0, 0, 0]
  Call Extruder 0.04526
  MoveL (T6497) to (121.16, 109.94, 8.3) mm, rotated rx 180 ry 0 rz -180 deg; joints [0, 0, 0, 0, 0, 0]
  Call Extruder 0.02915
  MoveL (T6498) to (121.16, 108.98, 8.3) mm, rotated rx 180 ry 0 rz -180 deg; joints [0, 0, 0, 0, 0, 0]
  Set speed (45.0 mm/s)
  Call Extruder -1.6
  MoveL (T6499) to (121.16, 108.98, 8.3) mm, rotated rx 180 ry 0 rz -180 deg; joints [0, 0, 0, 0, 0, 0]
  Set speed (120.0 mm/s)
  MoveL (T6500) to (121.16, 108.98, 8.3) mm, rotated rx 180 ry 0 rz -180 deg; joints [0, 0, 0, 0, 0, 0]
  Call Extruder -0.3409
  MoveL (T6501) to (121.16, 109.94, 8.3) mm, rotated rx 180 ry 0 rz -180 deg; joints [0, 0, 0, 0, 0, 0]
  Call Extruder -0.0391
  MoveL (T6502) to (121.05, 109.94, 8.3) mm, rotated rx 180 ry 0 rz -180 deg; joints [0, 0, 0, 0, 0, 0]
  Set speed (45.0 mm/s)
  Call Extruder -0.02
  MoveL (T6503) to (121.05, 109.94, 8.3) mm, rotated rx 180 ry 0 rz -180 deg; joints [0, 0, 0, 0, 0, 0]
  Set speed (150.0 mm/s)
  MoveL (T6504) to (121.05, 109.94, 10.3) mm, rotated rx 180 ry 0 rz -180 deg; joints [0, 0, 0, 0, 0, 0]
  MoveL (T6505) to (121.16, 115.5, 10.3) mm, rotated rx 180 ry 0 rz -180 deg; joints [0, 0, 0, 0, 0, 0]
  MoveL (T6506) to (121.16, 115.5, 8.3) mm, rotated rx 180 ry 0 rz -180 deg; joints [0, 0, 0, 0, 0, 0]
  Set speed (40.0 mm/s)
  Call Extruder 2.0
  MoveL (T6507) to (121.16, 115.5, 8.3) mm, rotated rx 180 ry 0 rz -180 deg; joints [0, 0, 0, 0, 0, 0]
  Set speed (25.0 mm/s)
  MoveL (T6508) to (121.16, 115.5, 8.3) mm, rotated rx 180 ry 0 rz -180 deg; joints [0, 0, 0, 0, 0, 0]
  Call Extruder 0.03633
  MoveL (T6509) to (121.16, 114.31, 8.3) mm, rotated rx 180 ry 0 rz -180 deg; joints [0, 0, 0, 0, 0, 0]
  Call Extruder 0.03807
  MoveL (T6510) to (119.91, 114.31, 8.3) mm, rotated rx 180 ry 0 rz -180 deg; joints [0, 0, 0, 0, 0, 0]
  Call Extruder 0.29512
  MoveL (T6511) to (113.06, 121.16, 8.3) mm, rotated rx 180 ry 0 rz -180 deg; joints [0, 0, 0, 0, 0, 0]
  Call Extruder 0.03385
  MoveL (T6512) to (111.94, 121.16, 8.3) mm, rotated rx 180 ry 0 rz -180 deg; joints [0, 0, 0, 0, 0, 0]
  Call Extruder 0.34896
  MoveL (T6513) to (103.84, 113.06, 8.3) mm, rotated rx 180 ry 0 rz -180 deg; joints [0, 0, 0, 0, 0, 0]
  Call Extruder 0.03385
  MoveL (T6514) to (103.84, 111.94, 8.3) mm, rotated rx 180 ry 0 rz -180 deg; joints [0, 0, 0, 0, 0, 0]
  Call Extruder 0.26732
  MoveL (T6515) to (110.05, 105.74, 8.3) mm, rotated rx 180 ry 0 rz -180 deg; joints [0, 0, 0, 0, 0, 0]
  Call Extruder 0.00901
  MoveL (T6516) to (110.34, 105.74, 8.3) mm, rotated rx 180 ry 0 rz -180 deg; joints [0, 0, 0, 0, 0, 0]
  Call Extruder 0.46574
  MoveL (T6517) to (121.16, 116.55, 8.3) mm, rotated rx 180 ry 0 rz -180 deg; joints [0, 0, 0, 0, 0, 0]
  Call Extruder 0.03385
  MoveL (T6518) to (121.16, 117.66, 8.3) mm, rotated rx 180 ry 0 rz -180 deg; joints [0, 0, 0, 0, 0, 0]
  Call Extruder 0.15054
  MoveL (T6519) to (117.66, 121.16, 8.3) mm, rotated rx 180 ry 0 rz -180 deg; joints [0, 0, 0, 0, 0, 0]
  Call Extruder 0.03385
  MoveL (T6520) to (116.55, 121.16, 8.3) mm, rotated rx 180 ry 0 rz -180 deg; joints [0, 0, 0, 0, 0, 0]
  Call Extruder 0.54738
  MoveL (T6521) to (103.84, 108.45, 8.3) mm, rotated rx 180 ry 0 rz -180 deg; joints [0, 0, 0, 0, 0, 0]
  Call Extruder 0.03385
  MoveL (T6522) to (103.84, 107.34, 8.3) mm, rotated rx 180 ry 0 rz -180 deg; joints [0, 0, 0, 0, 0, 0]
  Call Extruder 0.15054
  MoveL (T6523) to (107.34, 103.84, 8.3) mm, rotated rx 180 ry 0 rz -180 deg; joints [0, 0, 0, 0, 0, 0]
  Call Extruder 0.10645
  MoveL (T6524) to (103.84, 103.84, 8.3) mm, rotated rx 180 ry 0 rz -180 deg; joints [0, 0, 0, 0, 0, 0]
  Call Extruder 0.7458
  MoveL (T6525) to (121.16, 121.16, 8.3) mm, rotated rx 180 ry 0 rz -180 deg; joints [0, 0, 0, 0, 0, 0]
  Call Extruder 0.07441
  MoveL (T6526) to (118.71, 121.16, 8.3) mm, rotated rx 180 ry 0 rz -180 deg; joints [0, 0, 0, 0, 0, 0]
  Set speed (45.0 mm/s)
  Call Extruder -1.6
  MoveL (T6527) to (118.71, 121.16, 8.3) mm, rotated rx 180 ry 0 rz -180 deg; joints [0, 0, 0, 0, 0, 0]
  Set speed (120.0 mm/s)
  MoveL (T6528) to (118.71, 121.16, 8.3) mm, rotated rx 180 ry 0 rz -180 deg; joints [0, 0, 0, 0, 0, 0]
  Call Extruder -0.38
  MoveL (T6529) to (119.78, 121.16, 8.3) mm, rotated rx 180 ry 0 rz -180 deg; joints [0, 0, 0, 0, 0, 0]
  Set speed (45.0 mm/s)
  Call Extruder -0.02
  MoveL (T6530) to (119.78, 121.16, 8.3) mm, rotated rx 180 ry 0 rz -180 deg; joints [0, 0, 0, 0, 0, 0]
  Set speed (150.0 mm/s)
  MoveL (T6531) to (119.78, 121.16, 10.3) mm, rotated rx 180 ry 0 rz -180 deg; joints [0, 0, 0, 0, 0, 0]
  MoveL (T6532) to (104.34, 103.54, 10.3) mm, rotated rx 180 ry 0 rz -180 deg; joints [0, 0, 0, 0, 0, 0]
  MoveL (T6533) to (104.34, 103.54, 8.5) mm, rotated rx 180 ry 0 rz -180 deg; joints [0, 0, 0, 0, 0, 0]
  Set speed (40.0 mm/s)
  Call Extruder 2.0
  MoveL (T6534) to (104.34, 103.54, 8.5) mm, rotated rx 180 ry 0 rz -180 deg; joints [0, 0, 0, 0, 0, 0]
  Set speed (24.5 mm/s)
  MoveL (T6535) to (104.34, 103.54, 8.5) mm, rotated rx 180 ry 0 rz -180 deg; joints [0, 0, 0, 0, 0, 0]
  Call Extruder 0.14568
  MoveL (T6536) to (109.12, 103.54, 8.5) mm, rotated rx 180 ry 0 rz -180 deg; joints [0, 0, 0, 0, 0, 0]
  Call Extruder 0.05774
  MoveL (T6537) to (109.12, 105.43, 8.5) mm, rotated rx 180 ry 0 rz -180 deg; joints [0, 0, 0, 0, 0, 0]
  Call Extruder 0.17512
  MoveL (T6538) to (114.87, 105.43, 8.5) mm, rotated rx 180 ry 0 rz -180 deg; joints [0, 0, 0, 0, 0, 0]
  Call Extruder 0.05774
  MoveL (T6539) to (114.87, 103.54, 8.5) mm, rotated rx 180 ry 0 rz -180 deg; joints [0, 0, 0, 0, 0, 0]
  Call Extruder 0.20074
  MoveL (T6540) to (121.46, 103.54, 8.5) mm, rotated rx 180 ry 0 rz -180 deg; joints [0, 0, 0, 0, 0, 0]
  Call Extruder 0.20412
  MoveL (T6541) to (121.46, 110.24, 8.5) mm, rotated rx 180 ry 0 rz -180 deg; joints [0, 0, 0, 0, 0, 0]
  Call Extruder 0.05903
  MoveL (T6542) to (119.52, 110.24, 8.5) mm, rotated rx 180 ry 0 rz -180 deg; joints [0, 0, 0, 0, 0, 0]
  Call Extruder 0.11452
  MoveL (T6543) to (119.52, 114, 8.5) mm, rotated rx 180 ry 0 rz -180 deg; joints [0, 0, 0, 0, 0, 0]
  Call Extruder 0.05908
  MoveL (T6544) to (121.46, 114, 8.5) mm, rotated rx 180 ry 0 rz -180 deg; joints [0, 0, 0, 0, 0, 0]
  Call Extruder 0.22733
  MoveL (T6545) to (121.46, 121.46, 8.5) mm, rotated rx 180 ry 0 rz -180 deg; joints [0, 0, 0, 0, 0, 0]
  Call Extruder 0.54596
  MoveL (T6546) to (103.54, 121.46, 8.5) mm, rotated rx 180 ry 0 rz -180 deg; joints [0, 0, 0, 0, 0, 0]
  Call Extruder 0.54596
  MoveL (T6547) to (103.54, 103.54, 8.5) mm, rotated rx 180 ry 0 rz -180 deg; joints [0, 0, 0, 0, 0, 0]
  Call Extruder 0.02254
  MoveL (T6548) to (104.28, 103.54, 8.5) mm, rotated rx 180 ry 0 rz -180 deg; joints [0, 0, 0, 0, 0, 0]
  Set speed (150.0 mm/s)
  MoveL (T6549) to (103.53, 103.13, 8.5) mm, rotated rx 180 ry 0 rz -180 deg; joints [0, 0, 0, 0, 0, 0]
  Set speed (24.5 mm/s)
  MoveL (T6550) to (103.53, 103.13, 8.5) mm, rotated rx 180 ry 0 rz -180 deg; joints [0, 0, 0, 0, 0, 0]
  Call Extruder 0.18266
  MoveL (T6551) to (109.53, 103.13, 8.5) mm, rotated rx 180 ry 0 rz -180 deg; joints [0, 0, 0, 0, 0, 0]
  Call Extruder 0.05774
  MoveL (T6552) to (109.53, 105.03, 8.5) mm, rotated rx 180 ry 0 rz -180 deg; joints [0, 0, 0, 0, 0, 0]
  Call Extruder 0.15033
  MoveL (T6553) to (114.46, 105.03, 8.5) mm, rotated rx 180 ry 0 rz -180 deg; joints [0, 0, 0, 0, 0, 0]
  Call Extruder 0.05774
  MoveL (T6554) to (114.47, 103.13, 8.5) mm, rotated rx 180 ry 0 rz -180 deg; joints [0, 0, 0, 0, 0, 0]
  Call Extruder 0.22553
  MoveL (T6555) to (121.87, 103.13, 8.5) mm, rotated rx 180 ry 0 rz -180 deg; joints [0, 0, 0, 0, 0, 0]
  Call Extruder 0.22893
  MoveL (T6556) to (121.87, 110.65, 8.5) mm, rotated rx 180 ry 0 rz -180 deg; joints [0, 0, 0, 0, 0, 0]
  Call Extruder 0.05904
  MoveL (T6557) to (119.93, 110.65, 8.5) mm, rotated rx 180 ry 0 rz -180 deg; joints [0, 0, 0, 0, 0, 0]
  Call Extruder 0.08971
  MoveL (T6558) to (119.93, 113.59, 8.5) mm, rotated rx 180 ry 0 rz -180 deg; joints [0, 0, 0, 0, 0, 0]
  Call Extruder 0.05908
  MoveL (T6559) to (121.87, 113.59, 8.5) mm, rotated rx 180 ry 0 rz -180 deg; joints [0, 0, 0, 0, 0, 0]
  Call Extruder 0.25213
  MoveL (T6560) to (121.87, 121.87, 8.5) mm, rotated rx 180 ry 0 rz -180 deg; joints [0, 0, 0, 0, 0, 0]
  Call Extruder 0.57077
  MoveL (T6561) to (103.13, 121.87, 8.5) mm, rotated rx 180 ry 0 rz -180 deg; joints [0, 0, 0, 0, 0, 0]
  Call Extruder 0.57077
  MoveL (T6562) to (103.13, 103.13, 8.5) mm, rotated rx 180 ry 0 rz -180 deg; joints [0, 0, 0, 0, 0, 0]
  Call Extruder 0.01036
  MoveL (T6563) to (103.47, 103.13, 8.5) mm, rotated rx 180 ry 0 rz -180 deg; joints [0, 0, 0, 0, 0, 0]
  Set speed (150.0 mm/s)
  MoveL (T6564) to (102.72, 102.81, 8.5) mm, rotated rx 180 ry 0 rz -180 deg; joints [0, 0, 0, 0, 0, 0]
  Set speed (24.5 mm/s)
  MoveL (T6565) to (102.72, 102.81, 8.5) mm, rotated rx 180 ry 0 rz -180 deg; joints [0, 0, 0, 0, 0, 0]
  Call Extruder 0.00259
  MoveL (T6566) to (102.72, 102.72, 8.5) mm, rotated rx 180 ry 0 rz -180 deg; joints [0, 0, 0, 0, 0, 0]
  Call Extruder 0.21965
  MoveL (T6567) to (109.94, 102.72, 8.5) mm, rotated rx 180 ry 0 rz -180 deg; joints [0, 0, 0, 0, 0, 0]
  Call Extruder 0.05774
  MoveL (T6568) to (109.94, 104.62, 8.5) mm, rotated rx 180 ry 0 rz -180 deg; joints [0, 0, 0, 0, 0, 0]
  Call Extruder 0.12554
  MoveL (T6569) to (114.06, 104.62, 8.5) mm, rotated rx 180 ry 0 rz -180 deg; joints [0, 0, 0, 0, 0, 0]
  Call Extruder 0.05774
  MoveL (T6570) to (114.06, 102.72, 8.5) mm, rotated rx 180 ry 0 rz -180 deg; joints [0, 0, 0, 0, 0, 0]
  Call Extruder 0.25033
  MoveL (T6571) to (122.28, 102.72, 8.5) mm, rotated rx 180 ry 0 rz -180 deg; joints [0, 0, 0, 0, 0, 0]
  Call Extruder 0.25373
  MoveL (T6572) to (122.28, 111.05, 8.5) mm, rotated rx 180 ry 0 rz -180 deg; joints [0, 0, 0, 0, 0, 0]
  Call Extruder 0.05904
  MoveL (T6573) to (120.34, 111.05, 8.5) mm, rotated rx 180 ry 0 rz -180 deg; joints [0, 0, 0, 0, 0, 0]
  Call Extruder 0.06491
  MoveL (T6574) to (120.34, 113.18, 8.5) mm, rotated rx 180 ry 0 rz -180 deg; joints [0, 0, 0, 0, 0, 0]
  Call Extruder 0.05907
  MoveL (T6575) to (122.28, 113.19, 8.5) mm, rotated rx 180 ry 0 rz -180 deg; joints [0, 0, 0, 0, 0, 0]
  Call Extruder 0.27692
  MoveL (T6576) to (122.28, 122.28, 8.5) mm, rotated rx 180 ry 0 rz -180 deg; joints [0, 0, 0, 0, 0, 0]
  Call Extruder 0.59557
  MoveL (T6577) to (102.72, 122.28, 8.5) mm, rotated rx 180 ry 0 rz -180 deg; joints [0, 0, 0, 0, 0, 0]
  Call Extruder 0.59115
  MoveL (T6578) to (102.72, 102.87, 8.5) mm, rotated rx 180 ry 0 rz -180 deg; joints [0, 0, 0, 0, 0, 0]
  Set speed (150.0 mm/s)
  MoveL (T6579) to (102.78, 102.75, 8.5) mm, rotated rx 180 ry 0 rz -180 deg; joints [0, 0, 0, 0, 0, 0]
  Set speed (45.0 mm/s)
  Call Extruder -1.6
  MoveL (T6580) to (102.78, 102.75, 8.5) mm, rotated rx 180 ry 0 rz -180 deg; joints [0, 0, 0, 0, 0, 0]
  Set speed (120.0 mm/s)
  MoveL (T6581) to (102.78, 102.75, 8.5) mm, rotated rx 180 ry 0 rz -180 deg; joints [0, 0, 0, 0, 0, 0]
  Call Extruder -0.05166
  MoveL (T6582) to (102.72, 102.72, 8.5) mm, rotated rx 180 ry 0 rz -180 deg; joints [0, 0, 0, 0, 0, 0]
  Call Extruder -0.32834
  MoveL (T6583) to (103.65, 102.72, 8.5) mm, rotated rx 180 ry 0 rz -180 deg; joints [0, 0, 0, 0, 0, 0]
  Set speed (45.0 mm/s)
  Call Extruder -0.02
  MoveL (T6584) to (103.65, 102.72, 8.5) mm, rotated rx 180 ry 0 rz -180 deg; joints [0, 0, 0, 0, 0, 0]
  Set speed (150.0 mm/s)
  MoveL (T6585) to (103.65, 102.72, 10.5) mm, rotated rx 180 ry 0 rz -180 deg; joints [0, 0, 0, 0, 0, 0]
  MoveL (T6586) to (109, 104.69, 10.5) mm, rotated rx 180 ry 0 rz -180 deg; joints [0, 0, 0, 0, 0, 0]
  MoveL (T6587) to (109, 104.69, 8.5) mm, rotated rx 180 ry 0 rz -180 deg; joints [0, 0, 0, 0, 0, 0]
  Set speed (40.0 mm/s)
  Call Extruder 2.0
  MoveL (T6588) to (109, 104.69, 8.5) mm, rotated rx 180 ry 0 rz -180 deg; joints [0, 0, 0, 0, 0, 0]
  Set speed (24.5 mm/s)
  MoveL (T6589) to (109, 104.69, 8.5) mm, rotated rx 180 ry 0 rz -180 deg; joints [0, 0, 0, 0, 0, 0]
  Call Extruder 0.01598
  MoveL (T6590) to (108.65, 105.04, 8.5) mm, rotated rx 180 ry 0 rz -180 deg; joints [0, 0, 0, 0, 0, 0]
  Call Extruder 0.01988
  MoveL (T6591) to (108.65, 104.43, 8.5) mm, rotated rx 180 ry 0 rz -180 deg; joints [0, 0, 0, 0, 0, 0]
  Call Extruder 0.01598
  MoveL (T6592) to (109, 104.08, 8.5) mm, rotated rx 180 ry 0 rz -180 deg; joints [0, 0, 0, 0, 0, 0]
  Set speed (45.0 mm/s)
  Call Extruder -1.6
  MoveL (T6593) to (109, 104.08, 8.5) mm, rotated rx 180 ry 0 rz -180 deg; joints [0, 0, 0, 0, 0, 0]
  Set speed (120.0 mm/s)
  MoveL (T6594) to (109, 104.08, 8.5) mm, rotated rx 180 ry 0 rz -180 deg; joints [0, 0, 0, 0, 0, 0]
  Call Extruder -0.17547
  MoveL (T6595) to (108.65, 104.43, 8.5) mm, rotated rx 180 ry 0 rz -180 deg; joints [0, 0, 0, 0, 0, 0]
  Call Extruder -0.20453
  MoveL (T6596) to (108.65, 105, 8.5) mm, rotated rx 180 ry 0 rz -180 deg; joints [0, 0, 0, 0, 0, 0]
  Set speed (45.0 mm/s)
  Call Extruder -0.02
  MoveL (T6597) to (108.65, 105, 8.5) mm, rotated rx 180 ry 0 rz -180 deg; joints [0, 0, 0, 0, 0, 0]
  Set speed (150.0 mm/s)
  MoveL (T6598) to (108.65, 105, 10.5) mm, rotated rx 180 ry 0 rz -180 deg; joints [0, 0, 0, 0, 0, 0]
  MoveL (T6599) to (115.12, 105.64, 10.5) mm, rotated rx 180 ry 0 rz -180 deg; joints [0, 0, 0, 0, 0, 0]
  MoveL (T6600) to (115.12, 105.64, 8.5) mm, rotated rx 180 ry 0 rz -180 deg; joints [0, 0, 0, 0, 0, 0]
  Set speed (40.0 mm/s)
  Call Extruder 2.0
  MoveL (T6601) to (115.12, 105.64, 8.5) mm, rotated rx 180 ry 0 rz -180 deg; joints [0, 0, 0, 0, 0, 0]
  Set speed (24.5 mm/s)
  MoveL (T6602) to (115.12, 105.64, 8.5) mm, rotated rx 180 ry 0 rz -180 deg; joints [0, 0, 0, 0, 0, 0]
  Call Extruder 0.01303
  MoveL (T6603) to (115.4, 105.36, 8.5) mm, rotated rx 180 ry 0 rz -180 deg; joints [0, 0, 0, 0, 0, 0]
  Call Extruder 0.01996
  MoveL (T6604) to (115.4, 104.75, 8.5) mm, rotated rx 180 ry 0 rz -180 deg; joints [0, 0, 0, 0, 0, 0]
  Call Extruder 0.01044
  MoveL (T6605) to (115.18, 104.97, 8.5) mm, rotated rx 180 ry 0 rz -180 deg; joints [0, 0, 0, 0, 0, 0]
  Call Extruder 0.01996
  MoveL (T6606) to (115.18, 104.36, 8.5) mm, rotated rx 180 ry 0 rz -180 deg; joints [0, 0, 0, 0, 0, 0]
  Call Extruder 0.01886
  MoveL (T6607) to (115.59, 103.95, 8.5) mm, rotated rx 180 ry 0 rz -180 deg; joints [0, 0, 0, 0, 0, 0]
  Set speed (150.0 mm/s)
  MoveL (T6608) to (115.28, 105.87, 8.5) mm, rotated rx 180 ry 0 rz -180 deg; joints [0, 0, 0, 0, 0, 0]
  Set speed (24.5 mm/s)
  MoveL (T6609) to (115.28, 105.87, 8.5) mm, rotated rx 180 ry 0 rz -180 deg; joints [0, 0, 0, 0, 0, 0]
  Call Extruder 0.00635
  MoveL (T6610) to (115.49, 105.87, 8.5) mm, rotated rx 180 ry 0 rz -180 deg; joints [0, 0, 0, 0, 0, 0]
  Call Extruder 0.01375
  MoveL (T6611) to (115.81, 105.55, 8.5) mm, rotated rx 180 ry 0 rz -180 deg; joints [0, 0, 0, 0, 0, 0]
  Call Extruder 0.02936
  MoveL (T6612) to (115.81, 104.58, 8.5) mm, rotated rx 180 ry 0 rz -180 deg; joints [0, 0, 0, 0, 0, 0]
  Call Extruder 0.03186
  MoveL (T6613) to (116.55, 103.84, 8.5) mm, rotated rx 180 ry 0 rz -180 deg; joints [0, 0, 0, 0, 0, 0]
  Call Extruder 0.03385
  MoveL (T6614) to (117.66, 103.84, 8.5) mm, rotated rx 180 ry 0 rz -180 deg; joints [0, 0, 0, 0, 0, 0]
  Call Extruder 0.15054
  MoveL (T6615) to (121.16, 107.34, 8.5) mm, rotated rx 180 ry 0 rz -180 deg; joints [0, 0, 0, 0, 0, 0]
  Call Extruder 0.03385
  MoveL (T6616) to (121.16, 108.45, 8.5) mm, rotated rx 180 ry 0 rz -180 deg; joints [0, 0, 0, 0, 0, 0]
  Call Extruder 0.06391
  MoveL (T6617) to (119.67, 109.93, 8.5) mm, rotated rx 180 ry 0 rz -180 deg; joints [0, 0, 0, 0, 0, 0]
  Call Extruder 0.04519
  MoveL (T6618) to (121.16, 109.93, 8.5) mm, rotated rx 180 ry 0 rz -180 deg; joints [0, 0, 0, 0, 0, 0]
  Call Extruder 0.02922
  MoveL (T6619) to (121.16, 108.97, 8.5) mm, rotated rx 180 ry 0 rz -180 deg; joints [0, 0, 0, 0, 0, 0]
  Set speed (45.0 mm/s)
  Call Extruder -1.6
  MoveL (T6620) to (121.16, 108.97, 8.5) mm, rotated rx 180 ry 0 rz -180 deg; joints [0, 0, 0, 0, 0, 0]
  Set speed (120.0 mm/s)
  MoveL (T6621) to (121.16, 108.97, 8.5) mm, rotated rx 180 ry 0 rz -180 deg; joints [0, 0, 0, 0, 0, 0]
  Call Extruder -0.34167
  MoveL (T6622) to (121.16, 109.93, 8.5) mm, rotated rx 180 ry 0 rz -180 deg; joints [0, 0, 0, 0, 0, 0]
  Call Extruder -0.03833
  MoveL (T6623) to (121.05, 109.93, 8.5) mm, rotated rx 180 ry 0 rz -180 deg; joints [0, 0, 0, 0, 0, 0]
  Set speed (45.0 mm/s)
  Call Extruder -0.02
  MoveL (T6624) to (121.05, 109.93, 8.5) mm, rotated rx 180 ry 0 rz -180 deg; joints [0, 0, 0, 0, 0, 0]
  Set speed (150.0 mm/s)
  MoveL (T6625) to (121.05, 109.93, 10.5) mm, rotated rx 180 ry 0 rz -180 deg; joints [0, 0, 0, 0, 0, 0]
  MoveL (T6626) to (118.71, 103.84, 10.5) mm, rotated rx 180 ry 0 rz -180 deg; joints [0, 0, 0, 0, 0, 0]
  MoveL (T6627) to (118.71, 103.84, 8.5) mm, rotated rx 180 ry 0 rz -180 deg; joints [0, 0, 0, 0, 0, 0]
  Set speed (40.0 mm/s)
  Call Extruder 2.0
  MoveL (T6628) to (118.71, 103.84, 8.5) mm, rotated rx 180 ry 0 rz -180 deg; joints [0, 0, 0, 0, 0, 0]
  Set speed (24.5 mm/s)
  MoveL (T6629) to (118.71, 103.84, 8.5) mm, rotated rx 180 ry 0 rz -180 deg; joints [0, 0, 0, 0, 0, 0]
  Call Extruder 0.07441
  MoveL (T6630) to (121.16, 103.84, 8.5) mm, rotated rx 180 ry 0 rz -180 deg; joints [0, 0, 0, 0, 0, 0]
  Call Extruder 0.7458
  MoveL (T6631) to (103.84, 121.16, 8.5) mm, rotated rx 180 ry 0 rz -180 deg; joints [0, 0, 0, 0, 0, 0]
  Call Extruder 0.10645
  MoveL (T6632) to (103.84, 117.66, 8.5) mm, rotated rx 180 ry 0 rz -180 deg; joints [0, 0, 0, 0, 0, 0]
  Call Extruder 0.15054
  MoveL (T6633) to (107.34, 121.16, 8.5) mm, rotated rx 180 ry 0 rz -180 deg; joints [0, 0, 0, 0, 0, 0]
  Call Extruder 0.03385
  MoveL (T6634) to (108.45, 121.16, 8.5) mm, rotated rx 180 ry 0 rz -180 deg; joints [0, 0, 0, 0, 0, 0]
  Call Extruder 0.4639
  MoveL (T6635) to (119.22, 110.39, 8.5) mm, rotated rx 180 ry 0 rz -180 deg; joints [0, 0, 0, 0, 0, 0]
  Call Extruder 0.01161
  MoveL (T6636) to (119.22, 110.01, 8.5) mm, rotated rx 180 ry 0 rz -180 deg; joints [0, 0, 0, 0, 0, 0]
  Call Extruder 0.17832
  MoveL (T6637) to (115.08, 105.87, 8.5) mm, rotated rx 180 ry 0 rz -180 deg; joints [0, 0, 0, 0, 0, 0]
  Call Extruder 0.0036
  MoveL (T6638) to (114.96, 105.87, 8.5) mm, rotated rx 180 ry 0 rz -180 deg; joints [0, 0, 0, 0, 0, 0]
  Call Extruder 0.00552
  MoveL (T6639) to (114.83, 105.74, 8.5) mm, rotated rx 180 ry 0 rz -180 deg; joints [0, 0, 0, 0, 0, 0]
  Call Extruder 0.00541
  MoveL (T6640) to (114.66, 105.74, 8.5) mm, rotated rx 180 ry 0 rz -180 deg; joints [0, 0, 0, 0, 0, 0]
  Call Extruder 0.46573
  MoveL (T6641) to (103.84, 116.55, 8.5) mm, rotated rx 180 ry 0 rz -180 deg; joints [0, 0, 0, 0, 0, 0]
  Call Extruder 0.07441
  MoveL (T6642) to (103.84, 114.11, 8.5) mm, rotated rx 180 ry 0 rz -180 deg; joints [0, 0, 0, 0, 0, 0]
  Set speed (45.0 mm/s)
  Call Extruder -1.6
  MoveL (T6643) to (103.84, 114.11, 8.5) mm, rotated rx 180 ry 0 rz -180 deg; joints [0, 0, 0, 0, 0, 0]
  Set speed (120.0 mm/s)
  MoveL (T6644) to (103.84, 114.11, 8.5) mm, rotated rx 180 ry 0 rz -180 deg; joints [0, 0, 0, 0, 0, 0]
  Call Extruder -0.38
  MoveL (T6645) to (103.84, 115.17, 8.5) mm, rotated rx 180 ry 0 rz -180 deg; joints [0, 0, 0, 0, 0, 0]
  Set speed (45.0 mm/s)
  Call Extruder -0.02
  MoveL (T6646) to (103.84, 115.17, 8.5) mm, rotated rx 180 ry 0 rz -180 deg; joints [0, 0, 0, 0, 0, 0]
  Set speed (150.0 mm/s)
  MoveL (T6647) to (103.84, 115.17, 10.5) mm, rotated rx 180 ry 0 rz -180 deg; joints [0, 0, 0, 0, 0, 0]
  MoveL (T6648) to (118.71, 121.16, 10.5) mm, rotated rx 180 ry 0 rz -180 deg; joints [0, 0, 0, 0, 0, 0]
  MoveL (T6649) to (118.71, 121.16, 8.5) mm, rotated rx 180 ry 0 rz -180 deg; joints [0, 0, 0, 0, 0, 0]
  Set speed (40.0 mm/s)
  Call Extruder 2.0
  MoveL (T6650) to (118.71, 121.16, 8.5) mm, rotated rx 180 ry 0 rz -180 deg; joints [0, 0, 0, 0, 0, 0]
  Set speed (24.5 mm/s)
  MoveL (T6651) to (118.71, 121.16, 8.5) mm, rotated rx 180 ry 0 rz -180 deg; joints [0, 0, 0, 0, 0, 0]
  Call Extruder 0.07441
  MoveL (T6652) to (121.16, 121.16, 8.5) mm, rotated rx 180 ry 0 rz -180 deg; joints [0, 0, 0, 0, 0, 0]
  Call Extruder 0.7458
  MoveL (T6653) to (103.84, 103.84, 8.5) mm, rotated rx 180 ry 0 rz -180 deg; joints [0, 0, 0, 0, 0, 0]
  Call Extruder 0.10645
  MoveL (T6654) to (107.34, 103.84, 8.5) mm, rotated rx 180 ry 0 rz -180 deg; joints [0, 0, 0, 0, 0, 0]
  Call Extruder 0.15054
  MoveL (T6655) to (103.84, 107.34, 8.5) mm, rotated rx 180 ry 0 rz -180 deg; joints [0, 0, 0, 0, 0, 0]
  Call Extruder 0.03385
  MoveL (T6656) to (103.84, 108.45, 8.5) mm, rotated rx 180 ry 0 rz -180 deg; joints [0, 0, 0, 0, 0, 0]
  Call Extruder 0.54738
  MoveL (T6657) to (116.55, 121.16, 8.5) mm, rotated rx 180 ry 0 rz -180 deg; joints [0, 0, 0, 0, 0, 0]
  Call Extruder 0.03385
  MoveL (T6658) to (117.66, 121.16, 8.5) mm, rotated rx 180 ry 0 rz -180 deg; joints [0, 0, 0, 0, 0, 0]
  Call Extruder 0.15054
  MoveL (T6659) to (121.16, 117.66, 8.5) mm, rotated rx 180 ry 0 rz -180 deg; joints [0, 0, 0, 0, 0, 0]
  Call Extruder 0.03385
  MoveL (T6660) to (121.16, 116.55, 8.5) mm, rotated rx 180 ry 0 rz -180 deg; joints [0, 0, 0, 0, 0, 0]
  Call Extruder 0.46573
  MoveL (T6661) to (110.34, 105.74, 8.5) mm, rotated rx 180 ry 0 rz -180 deg; joints [0, 0, 0, 0, 0, 0]
  Call Extruder 0.00902
  MoveL (T6662) to (110.05, 105.74, 8.5) mm, rotated rx 180 ry 0 rz -180 deg; joints [0, 0, 0, 0, 0, 0]
  Call Extruder 0.26731
  MoveL (T6663) to (103.84, 111.94, 8.5) mm, rotated rx 180 ry 0 rz -180 deg; joints [0, 0, 0, 0, 0, 0]
  Call Extruder 0.03385
  MoveL (T6664) to (103.84, 113.06, 8.5) mm, rotated rx 180 ry 0 rz -180 deg; joints [0, 0, 0, 0, 0, 0]
  Call Extruder 0.34896
  MoveL (T6665) to (111.94, 121.16, 8.5) mm, rotated rx 180 ry 0 rz -180 deg; joints [0, 0, 0, 0, 0, 0]
  Call Extruder 0.03385
  MoveL (T6666) to (113.06, 121.16, 8.5) mm, rotated rx 180 ry 0 rz -180 deg; joints [0, 0, 0, 0, 0, 0]
  Call Extruder 0.29521
  MoveL (T6667) to (119.91, 114.3, 8.5) mm, rotated rx 180 ry 0 rz -180 deg; joints [0, 0, 0, 0, 0, 0]
  Call Extruder 0.03801
  MoveL (T6668) to (121.16, 114.3, 8.5) mm, rotated rx 180 ry 0 rz -180 deg; joints [0, 0, 0, 0, 0, 0]
  Call Extruder 0.0364
  MoveL (T6669) to (121.16, 115.5, 8.5) mm, rotated rx 180 ry 0 rz -180 deg; joints [0, 0, 0, 0, 0, 0]
  Set speed (45.0 mm/s)
  Call Extruder -1.6
  MoveL (T6670) to (121.16, 115.5, 8.5) mm, rotated rx 180 ry 0 rz -180 deg; joints [0, 0, 0, 0, 0, 0]
  Set speed (120.0 mm/s)
  MoveL (T6671) to (121.16, 115.5, 8.5) mm, rotated rx 180 ry 0 rz -180 deg; joints [0, 0, 0, 0, 0, 0]
  Call Extruder -0.38
  MoveL (T6672) to (121.16, 114.43, 8.5) mm, rotated rx 180 ry 0 rz -180 deg; joints [0, 0, 0, 0, 0, 0]
  Set speed (45.0 mm/s)
  Call Extruder -0.02
  MoveL (T6673) to (121.16, 114.43, 8.5) mm, rotated rx 180 ry 0 rz -180 deg; joints [0, 0, 0, 0, 0, 0]
  Set speed (150.0 mm/s)
  MoveL (T6674) to (121.16, 114.43, 10.5) mm, rotated rx 180 ry 0 rz -180 deg; joints [0, 0, 0, 0, 0, 0]
  MoveL (T6675) to (104.34, 103.54, 10.5) mm, rotated rx 180 ry 0 rz -180 deg; joints [0, 0, 0, 0, 0, 0]
  MoveL (T6676) to (104.34, 103.54, 8.7) mm, rotated rx 180 ry 0 rz -180 deg; joints [0, 0, 0, 0, 0, 0]
  Set speed (40.0 mm/s)
  Call Extruder 2.0
  MoveL (T6677) to (104.34, 103.54, 8.7) mm, rotated rx 180 ry 0 rz -180 deg; joints [0, 0, 0, 0, 0, 0]
  Set speed (24.5 mm/s)
  MoveL (T6678) to (104.34, 103.54, 8.7) mm, rotated rx 180 ry 0 rz -180 deg; joints [0, 0, 0, 0, 0, 0]
  Call Extruder 0.14906
  MoveL (T6679) to (109.23, 103.54, 8.7) mm, rotated rx 180 ry 0 rz -180 deg; joints [0, 0, 0, 0, 0, 0]
  Call Extruder 0.05774
  MoveL (T6680) to (109.23, 105.44, 8.7) mm, rotated rx 180 ry 0 rz -180 deg; joints [0, 0, 0, 0, 0, 0]
  Call Extruder 0.16788
  MoveL (T6681) to (114.74, 105.44, 8.7) mm, rotated rx 180 ry 0 rz -180 deg; joints [0, 0, 0, 0, 0, 0]
  Call Extruder 0.05774
  MoveL (T6682) to (114.75, 103.54, 8.7) mm, rotated rx 180 ry 0 rz -180 deg; joints [0, 0, 0, 0, 0, 0]
  Call Extruder 0.20459
  MoveL (T6683) to (121.46, 103.54, 8.7) mm, rotated rx 180 ry 0 rz -180 deg; joints [0, 0, 0, 0, 0, 0]
  Call Extruder 0.20405
  MoveL (T6684) to (121.46, 110.24, 8.7) mm, rotated rx 180 ry 0 rz -180 deg; joints [0, 0, 0, 0, 0, 0]
  Call Extruder 0.05902
  MoveL (T6685) to (119.52, 110.24, 8.7) mm, rotated rx 180 ry 0 rz -180 deg; joints [0, 0, 0, 0, 0, 0]
  Call Extruder 0.11452
  MoveL (T6686) to (119.52, 114, 8.7) mm, rotated rx 180 ry 0 rz -180 deg; joints [0, 0, 0, 0, 0, 0]
  Call Extruder 0.05907
  MoveL (T6687) to (121.46, 114, 8.7) mm, rotated rx 180 ry 0 rz -180 deg; joints [0, 0, 0, 0, 0, 0]
  Call Extruder 0.22739
  MoveL (T6688) to (121.46, 121.46, 8.7) mm, rotated rx 180 ry 0 rz -180 deg; joints [0, 0, 0, 0, 0, 0]
  Call Extruder 0.54596
  MoveL (T6689) to (103.54, 121.46, 8.7) mm, rotated rx 180 ry 0 rz -180 deg; joints [0, 0, 0, 0, 0, 0]
  Call Extruder 0.54596
  MoveL (T6690) to (103.54, 103.54, 8.7) mm, rotated rx 180 ry 0 rz -180 deg; joints [0, 0, 0, 0, 0, 0]
  Call Extruder 0.02254
  MoveL (T6691) to (104.28, 103.54, 8.7) mm, rotated rx 180 ry 0 rz -180 deg; joints [0, 0, 0, 0, 0, 0]
  Set speed (150.0 mm/s)
  MoveL (T6692) to (103.53, 103.13, 8.7) mm, rotated rx 180 ry 0 rz -180 deg; joints [0, 0, 0, 0, 0, 0]
  Set speed (24.5 mm/s)
  MoveL (T6693) to (103.53, 103.13, 8.7) mm, rotated rx 180 ry 0 rz -180 deg; joints [0, 0, 0, 0, 0, 0]
  Call Extruder 0.18605
  MoveL (T6694) to (109.64, 103.13, 8.7) mm, rotated rx 180 ry 0 rz -180 deg; joints [0, 0, 0, 0, 0, 0]
  Call Extruder 0.05774
  MoveL (T6695) to (109.64, 105.03, 8.7) mm, rotated rx 180 ry 0 rz -180 deg; joints [0, 0, 0, 0, 0, 0]
  Call Extruder 0.14309
  MoveL (T6696) to (114.34, 105.03, 8.7) mm, rotated rx 180 ry 0 rz -180 deg; joints [0, 0, 0, 0, 0, 0]
  Call Extruder 0.05774
  MoveL (T6697) to (114.34, 103.13, 8.7) mm, rotated rx 180 ry 0 rz -180 deg; joints [0, 0, 0, 0, 0, 0]
  Call Extruder 0.22938
  MoveL (T6698) to (121.87, 103.13, 8.7) mm, rotated rx 180 ry 0 rz -180 deg; joints [0, 0, 0, 0, 0, 0]
  Call Extruder 0.22886
  MoveL (T6699) to (121.87, 110.64, 8.7) mm, rotated rx 180 ry 0 rz -180 deg; joints [0, 0, 0, 0, 0, 0]
  Call Extruder 0.05903
  MoveL (T6700) to (119.93, 110.64, 8.7) mm, rotated rx 180 ry 0 rz -180 deg; joints [0, 0, 0, 0, 0, 0]
  Call Extruder 0.08971
  MoveL (T6701) to (119.93, 113.59, 8.7) mm, rotated rx 180 ry 0 rz -180 deg; joints [0, 0, 0, 0, 0, 0]
  Call Extruder 0.05907
  MoveL (T6702) to (121.87, 113.59, 8.7) mm, rotated rx 180 ry 0 rz -180 deg; joints [0, 0, 0, 0, 0, 0]
  Call Extruder 0.25219
  MoveL (T6703) to (121.87, 121.87, 8.7) mm, rotated rx 180 ry 0 rz -180 deg; joints [0, 0, 0, 0, 0, 0]
  Call Extruder 0.57077
  MoveL (T6704) to (103.13, 121.87, 8.7) mm, rotated rx 180 ry 0 rz -180 deg; joints [0, 0, 0, 0, 0, 0]
  Call Extruder 0.57077
  MoveL (T6705) to (103.13, 103.13, 8.7) mm, rotated rx 180 ry 0 rz -180 deg; joints [0, 0, 0, 0, 0, 0]
  Call Extruder 0.01036
  MoveL (T6706) to (103.47, 103.13, 8.7) mm, rotated rx 180 ry 0 rz -180 deg; joints [0, 0, 0, 0, 0, 0]
  Set speed (150.0 mm/s)
  MoveL (T6707) to (102.72, 102.81, 8.7) mm, rotated rx 180 ry 0 rz -180 deg; joints [0, 0, 0, 0, 0, 0]
  Set speed (24.5 mm/s)
  MoveL (T6708) to (102.72, 102.81, 8.7) mm, rotated rx 180 ry 0 rz -180 deg; joints [0, 0, 0, 0, 0, 0]
  Call Extruder 0.00259
  MoveL (T6709) to (102.72, 102.72, 8.7) mm, rotated rx 180 ry 0 rz -180 deg; joints [0, 0, 0, 0, 0, 0]
  Call Extruder 0.22303
  MoveL (T6710) to (110.05, 102.72, 8.7) mm, rotated rx 180 ry 0 rz -180 deg; joints [0, 0, 0, 0, 0, 0]
  Call Extruder 0.05774
  MoveL (T6711) to (110.05, 104.62, 8.7) mm, rotated rx 180 ry 0 rz -180 deg; joints [0, 0, 0, 0, 0, 0]
  Call Extruder 0.1183
  MoveL (T6712) to (113.93, 104.62, 8.7) mm, rotated rx 180 ry 0 rz -180 deg; joints [0, 0, 0, 0, 0, 0]
  Call Extruder 0.05774
  MoveL (T6713) to (113.93, 102.72, 8.7) mm, rotated rx 180 ry 0 rz -180 deg; joints [0, 0, 0, 0, 0, 0]
  Call Extruder 0.25418
  MoveL (T6714) to (122.28, 102.72, 8.7) mm, rotated rx 180 ry 0 rz -180 deg; joints [0, 0, 0, 0, 0, 0]
  Call Extruder 0.25367
  MoveL (T6715) to (122.28, 111.05, 8.7) mm, rotated rx 180 ry 0 rz -180 deg; joints [0, 0, 0, 0, 0, 0]
  Call Extruder 0.05903
  MoveL (T6716) to (120.34, 111.05, 8.7) mm, rotated rx 180 ry 0 rz -180 deg; joints [0, 0, 0, 0, 0, 0]
  Call Extruder 0.06491
  MoveL (T6717) to (120.34, 113.18, 8.7) mm, rotated rx 180 ry 0 rz -180 deg; joints [0, 0, 0, 0, 0, 0]
  Call Extruder 0.05906
  MoveL (T6718) to (122.28, 113.18, 8.7) mm, rotated rx 180 ry 0 rz -180 deg; joints [0, 0, 0, 0, 0, 0]
  Call Extruder 0.27699
  MoveL (T6719) to (122.28, 122.28, 8.7) mm, rotated rx 180 ry 0 rz -180 deg; joints [0, 0, 0, 0, 0, 0]
  Call Extruder 0.59557
  MoveL (T6720) to (102.72, 122.28, 8.7) mm, rotated rx 180 ry 0 rz -180 deg; joints [0, 0, 0, 0, 0, 0]
  Call Extruder 0.59115
  MoveL (T6721) to (102.72, 102.87, 8.7) mm, rotated rx 180 ry 0 rz -180 deg; joints [0, 0, 0, 0, 0, 0]
  Set speed (150.0 mm/s)
  MoveL (T6722) to (102.78, 102.75, 8.7) mm, rotated rx 180 ry 0 rz -180 deg; joints [0, 0, 0, 0, 0, 0]
  Set speed (45.0 mm/s)
  Call Extruder -1.6
  MoveL (T6723) to (102.78, 102.75, 8.7) mm, rotated rx 180 ry 0 rz -180 deg; joints [0, 0, 0, 0, 0, 0]
  Set speed (120.0 mm/s)
  MoveL (T6724) to (102.78, 102.75, 8.7) mm, rotated rx 180 ry 0 rz -180 deg; joints [0, 0, 0, 0, 0, 0]
  Call Extruder -0.05166
  MoveL (T6725) to (102.72, 102.72, 8.7) mm, rotated rx 180 ry 0 rz -180 deg; joints [0, 0, 0, 0, 0, 0]
  Call Extruder -0.32834
  MoveL (T6726) to (103.65, 102.72, 8.7) mm, rotated rx 180 ry 0 rz -180 deg; joints [0, 0, 0, 0, 0, 0]
  Set speed (45.0 mm/s)
  Call Extruder -0.02
  MoveL (T6727) to (103.65, 102.72, 8.7) mm, rotated rx 180 ry 0 rz -180 deg; joints [0, 0, 0, 0, 0, 0]
  Set speed (150.0 mm/s)
  MoveL (T6728) to (103.65, 102.72, 10.7) mm, rotated rx 180 ry 0 rz -180 deg; joints [0, 0, 0, 0, 0, 0]
  MoveL (T6729) to (108.58, 103.99, 10.7) mm, rotated rx 180 ry 0 rz -180 deg; joints [0, 0, 0, 0, 0, 0]
  MoveL (T6730) to (108.58, 103.99, 8.7) mm, rotated rx 180 ry 0 rz -180 deg; joints [0, 0, 0, 0, 0, 0]
  Set speed (40.0 mm/s)
  Call Extruder 2.0
  MoveL (T6731) to (108.58, 103.99, 8.7) mm, rotated rx 180 ry 0 rz -180 deg; joints [0, 0, 0, 0, 0, 0]
  Set speed (24.5 mm/s)
  MoveL (T6732) to (108.58, 103.99, 8.7) mm, rotated rx 180 ry 0 rz -180 deg; joints [0, 0, 0, 0, 0, 0]
  Call Extruder 0.01562
  MoveL (T6733) to (108.93, 104.34, 8.7) mm, rotated rx 180 ry 0 rz -180 deg; joints [0, 0, 0, 0, 0, 0]
  Call Extruder 0.01897
  MoveL (T6734) to (108.93, 104.94, 8.7) mm, rotated rx 180 ry 0 rz -180 deg; joints [0, 0, 0, 0, 0, 0]
  Call Extruder 0.00741
  MoveL (T6735) to (108.76, 104.77, 8.7) mm, rotated rx 180 ry 0 rz -180 deg; joints [0, 0, 0, 0, 0, 0]
  Call Extruder 0.01897
  MoveL (T6736) to (108.76, 105.37, 8.7) mm, rotated rx 180 ry 0 rz -180 deg; joints [0, 0, 0, 0, 0, 0]
  Call Extruder 0.01235
  MoveL (T6737) to (109.04, 105.64, 8.7) mm, rotated rx 180 ry 0 rz -180 deg; joints [0, 0, 0, 0, 0, 0]
  Set speed (45.0 mm/s)
  Call Extruder -1.6
  MoveL (T6738) to (109.04, 105.64, 8.7) mm, rotated rx 180 ry 0 rz -180 deg; joints [0, 0, 0, 0, 0, 0]
  Set speed (120.0 mm/s)
  MoveL (T6739) to (109.04, 105.64, 8.7) mm, rotated rx 180 ry 0 rz -180 deg; joints [0, 0, 0, 0, 0, 0]
  Call Extruder -0.13884
  MoveL (T6740) to (108.76, 105.37, 8.7) mm, rotated rx 180 ry 0 rz -180 deg; joints [0, 0, 0, 0, 0, 0]
  Call Extruder -0.21338
  MoveL (T6741) to (108.76, 104.77, 8.7) mm, rotated rx 180 ry 0 rz -180 deg; joints [0, 0, 0, 0, 0, 0]
  Call Extruder -0.02778
  MoveL (T6742) to (108.82, 104.83, 8.7) mm, rotated rx 180 ry 0 rz -180 deg; joints [0, 0, 0, 0, 0, 0]
  Set speed (45.0 mm/s)
  Call Extruder -0.02
  MoveL (T6743) to (108.82, 104.83, 8.7) mm, rotated rx 180 ry 0 rz -180 deg; joints [0, 0, 0, 0, 0, 0]
  Set speed (150.0 mm/s)
  MoveL (T6744) to (108.82, 104.83, 10.7) mm, rotated rx 180 ry 0 rz -180 deg; joints [0, 0, 0, 0, 0, 0]
  MoveL (T6745) to (115.46, 104.64, 10.7) mm, rotated rx 180 ry 0 rz -180 deg; joints [0, 0, 0, 0, 0, 0]
  MoveL (T6746) to (115.46, 104.64, 8.7) mm, rotated rx 180 ry 0 rz -180 deg; joints [0, 0, 0, 0, 0, 0]
  Set speed (40.0 mm/s)
  Call Extruder 2.0
  MoveL (T6747) to (115.46, 104.64, 8.7) mm, rotated rx 180 ry 0 rz -180 deg; joints [0, 0, 0, 0, 0, 0]
  Set speed (24.5 mm/s)
  MoveL (T6748) to (115.46, 104.64, 8.7) mm, rotated rx 180 ry 0 rz -180 deg; joints [0, 0, 0, 0, 0, 0]
  Call Extruder 0.01928
  MoveL (T6749) to (115.05, 104.22, 8.7) mm, rotated rx 180 ry 0 rz -180 deg; joints [0, 0, 0, 0, 0, 0]
  Call Extruder 0.02089
  MoveL (T6750) to (115.05, 104.85, 8.7) mm, rotated rx 180 ry 0 rz -180 deg; joints [0, 0, 0, 0, 0, 0]
  Call Extruder 0.01928
  MoveL (T6751) to (115.46, 105.26, 8.7) mm, rotated rx 180 ry 0 rz -180 deg; joints [0, 0, 0, 0, 0, 0]
  Set speed (150.0 mm/s)
  MoveL (T6752) to (116.35, 103.84, 8.7) mm, rotated rx 180 ry 0 rz -180 deg; joints [0, 0, 0, 0, 0, 0]
  Set speed (24.5 mm/s)
  MoveL (T6753) to (116.35, 103.84, 8.7) mm, rotated rx 180 ry 0 rz -180 deg; joints [0, 0, 0, 0, 0, 0]
  Call Extruder 0.02017
  MoveL (T6754) to (115.68, 103.84, 8.7) mm, rotated rx 180 ry 0 rz -180 deg; joints [0, 0, 0, 0, 0, 0]
  Call Extruder 0.02638
  MoveL (T6755) to (115.68, 104.71, 8.7) mm, rotated rx 180 ry 0 rz -180 deg; joints [0, 0, 0, 0, 0, 0]
  Call Extruder 0.03731
  MoveL (T6756) to (116.55, 103.84, 8.7) mm, rotated rx 180 ry 0 rz -180 deg; joints [0, 0, 0, 0, 0, 0]
  Call Extruder 0.03385
  MoveL (T6757) to (117.66, 103.84, 8.7) mm, rotated rx 180 ry 0 rz -180 deg; joints [0, 0, 0, 0, 0, 0]
  Call Extruder 0.15054
  MoveL (T6758) to (121.16, 107.34, 8.7) mm, rotated rx 180 ry 0 rz -180 deg; joints [0, 0, 0, 0, 0, 0]
  Call Extruder 0.03385
  MoveL (T6759) to (121.16, 108.45, 8.7) mm, rotated rx 180 ry 0 rz -180 deg; joints [0, 0, 0, 0, 0, 0]
  Call Extruder 0.06381
  MoveL (T6760) to (119.67, 109.93, 8.7) mm, rotated rx 180 ry 0 rz -180 deg; joints [0, 0, 0, 0, 0, 0]
  Call Extruder 0.04512
  MoveL (T6761) to (121.16, 109.93, 8.7) mm, rotated rx 180 ry 0 rz -180 deg; joints [0, 0, 0, 0, 0, 0]
  Call Extruder 0.02928
  MoveL (T6762) to (121.16, 108.97, 8.7) mm, rotated rx 180 ry 0 rz -180 deg; joints [0, 0, 0, 0, 0, 0]
  Set speed (45.0 mm/s)
  Call Extruder -1.6
  MoveL (T6763) to (121.16, 108.97, 8.7) mm, rotated rx 180 ry 0 rz -180 deg; joints [0, 0, 0, 0, 0, 0]
  Set speed (120.0 mm/s)
  MoveL (T6764) to (121.16, 108.97, 8.7) mm, rotated rx 180 ry 0 rz -180 deg; joints [0, 0, 0, 0, 0, 0]
  Call Extruder -0.34245
  MoveL (T6765) to (121.16, 109.93, 8.7) mm, rotated rx 180 ry 0 rz -180 deg; joints [0, 0, 0, 0, 0, 0]
  Call Extruder -0.03755
  MoveL (T6766) to (121.05, 109.93, 8.7) mm, rotated rx 180 ry 0 rz -180 deg; joints [0, 0, 0, 0, 0, 0]
  Set speed (45.0 mm/s)
  Call Extruder -0.02
  MoveL (T6767) to (121.05, 109.93, 8.7) mm, rotated rx 180 ry 0 rz -180 deg; joints [0, 0, 0, 0, 0, 0]
  Set speed (150.0 mm/s)
  MoveL (T6768) to (121.05, 109.93, 10.7) mm, rotated rx 180 ry 0 rz -180 deg; joints [0, 0, 0, 0, 0, 0]
  MoveL (T6769) to (118.71, 103.84, 10.7) mm, rotated rx 180 ry 0 rz -180 deg; joints [0, 0, 0, 0, 0, 0]
  MoveL (T6770) to (118.71, 103.84, 8.7) mm, rotated rx 180 ry 0 rz -180 deg; joints [0, 0, 0, 0, 0, 0]
  Set speed (40.0 mm/s)
  Call Extruder 2.0
  MoveL (T6771) to (118.71, 103.84, 8.7) mm, rotated rx 180 ry 0 rz -180 deg; joints [0, 0, 0, 0, 0, 0]
  Set speed (24.5 mm/s)
  MoveL (T6772) to (118.71, 103.84, 8.7) mm, rotated rx 180 ry 0 rz -180 deg; joints [0, 0, 0, 0, 0, 0]
  Call Extruder 0.07441
  MoveL (T6773) to (121.16, 103.84, 8.7) mm, rotated rx 180 ry 0 rz -180 deg; joints [0, 0, 0, 0, 0, 0]
  Call Extruder 0.7458
  MoveL (T6774) to (103.84, 121.16, 8.7) mm, rotated rx 180 ry 0 rz -180 deg; joints [0, 0, 0, 0, 0, 0]
  Call Extruder 0.10645
  MoveL (T6775) to (103.84, 117.66, 8.7) mm, rotated rx 180 ry 0 rz -180 deg; joints [0, 0, 0, 0, 0, 0]
  Call Extruder 0.15054
  MoveL (T6776) to (107.34, 121.16, 8.7) mm, rotated rx 180 ry 0 rz -180 deg; joints [0, 0, 0, 0, 0, 0]
  Call Extruder 0.03385
  MoveL (T6777) to (108.45, 121.16, 8.7) mm, rotated rx 180 ry 0 rz -180 deg; joints [0, 0, 0, 0, 0, 0]
  Call Extruder 0.46391
  MoveL (T6778) to (119.22, 110.39, 8.7) mm, rotated rx 180 ry 0 rz -180 deg; joints [0, 0, 0, 0, 0, 0]
  Call Extruder 0.01159
  MoveL (T6779) to (119.22, 110.01, 8.7) mm, rotated rx 180 ry 0 rz -180 deg; joints [0, 0, 0, 0, 0, 0]
  Call Extruder 0.17833
  MoveL (T6780) to (115.08, 105.87, 8.7) mm, rotated rx 180 ry 0 rz -180 deg; joints [0, 0, 0, 0, 0, 0]
  Call Extruder 0.00745
  MoveL (T6781) to (114.83, 105.87, 8.7) mm, rotated rx 180 ry 0 rz -180 deg; joints [0, 0, 0, 0, 0, 0]
  Call Extruder 0.00552
  MoveL (T6782) to (114.71, 105.74, 8.7) mm, rotated rx 180 ry 0 rz -180 deg; joints [0, 0, 0, 0, 0, 0]
  Call Extruder 0.00157
  MoveL (T6783) to (114.66, 105.74, 8.7) mm, rotated rx 180 ry 0 rz -180 deg; joints [0, 0, 0, 0, 0, 0]
  Call Extruder 0.46572
  MoveL (T6784) to (103.84, 116.55, 8.7) mm, rotated rx 180 ry 0 rz -180 deg; joints [0, 0, 0, 0, 0, 0]
  Call Extruder 0.07441
  MoveL (T6785) to (103.84, 114.11, 8.7) mm, rotated rx 180 ry 0 rz -180 deg; joints [0, 0, 0, 0, 0, 0]
  Set speed (45.0 mm/s)
  Call Extruder -1.6
  MoveL (T6786) to (103.84, 114.11, 8.7) mm, rotated rx 180 ry 0 rz -180 deg; joints [0, 0, 0, 0, 0, 0]
  Set speed (120.0 mm/s)
  MoveL (T6787) to (103.84, 114.11, 8.7) mm, rotated rx 180 ry 0 rz -180 deg; joints [0, 0, 0, 0, 0, 0]
  Call Extruder -0.38
  MoveL (T6788) to (103.84, 115.17, 8.7) mm, rotated rx 180 ry 0 rz -180 deg; joints [0, 0, 0, 0, 0, 0]
  Set speed (45.0 mm/s)
  Call Extruder -0.02
  MoveL (T6789) to (103.84, 115.17, 8.7) mm, rotated rx 180 ry 0 rz -180 deg; joints [0, 0, 0, 0, 0, 0]
  Set speed (150.0 mm/s)
  MoveL (T6790) to (103.84, 115.17, 10.7) mm, rotated rx 180 ry 0 rz -180 deg; joints [0, 0, 0, 0, 0, 0]
  MoveL (T6791) to (118.71, 121.16, 10.7) mm, rotated rx 180 ry 0 rz -180 deg; joints [0, 0, 0, 0, 0, 0]
  MoveL (T6792) to (118.71, 121.16, 8.7) mm, rotated rx 180 ry 0 rz -180 deg; joints [0, 0, 0, 0, 0, 0]
  Set speed (40.0 mm/s)
  Call Extruder 2.0
  MoveL (T6793) to (118.71, 121.16, 8.7) mm, rotated rx 180 ry 0 rz -180 deg; joints [0, 0, 0, 0, 0, 0]
  Set speed (24.5 mm/s)
  MoveL (T6794) to (118.71, 121.16, 8.7) mm, rotated rx 180 ry 0 rz -180 deg; joints [0, 0, 0, 0, 0, 0]
  Call Extruder 0.07441
  MoveL (T6795) to (121.16, 121.16, 8.7) mm, rotated rx 180 ry 0 rz -180 deg; joints [0, 0, 0, 0, 0, 0]
  Call Extruder 0.7458
  MoveL (T6796) to (103.84, 103.84, 8.7) mm, rotated rx 180 ry 0 rz -180 deg; joints [0, 0, 0, 0, 0, 0]
  Call Extruder 0.10645
  MoveL (T6797) to (107.34, 103.84, 8.7) mm, rotated rx 180 ry 0 rz -180 deg; joints [0, 0, 0, 0, 0, 0]
  Call Extruder 0.15054
  MoveL (T6798) to (103.84, 107.34, 8.7) mm, rotated rx 180 ry 0 rz -180 deg; joints [0, 0, 0, 0, 0, 0]
  Call Extruder 0.03385
  MoveL (T6799) to (103.84, 108.45, 8.7) mm, rotated rx 180 ry 0 rz -180 deg; joints [0, 0, 0, 0, 0, 0]
  Call Extruder 0.54738
  MoveL (T6800) to (116.55, 121.16, 8.7) mm, rotated rx 180 ry 0 rz -180 deg; joints [0, 0, 0, 0, 0, 0]
  Call Extruder 0.03385
  MoveL (T6801) to (117.66, 121.16, 8.7) mm, rotated rx 180 ry 0 rz -180 deg; joints [0, 0, 0, 0, 0, 0]
  Call Extruder 0.15054
  MoveL (T6802) to (121.16, 117.66, 8.7) mm, rotated rx 180 ry 0 rz -180 deg; joints [0, 0, 0, 0, 0, 0]
  Call Extruder 0.03385
  MoveL (T6803) to (121.16, 116.55, 8.7) mm, rotated rx 180 ry 0 rz -180 deg; joints [0, 0, 0, 0, 0, 0]
  Call Extruder 0.46572
  MoveL (T6804) to (110.34, 105.74, 8.7) mm, rotated rx 180 ry 0 rz -180 deg; joints [0, 0, 0, 0, 0, 0]
  Call Extruder 0.00903
  MoveL (T6805) to (110.05, 105.74, 8.7) mm, rotated rx 180 ry 0 rz -180 deg; joints [0, 0, 0, 0, 0, 0]
  Call Extruder 0.2673
  MoveL (T6806) to (103.84, 111.94, 8.7) mm, rotated rx 180 ry 0 rz -180 deg; joints [0, 0, 0, 0, 0, 0]
  Call Extruder 0.03385
  MoveL (T6807) to (103.84, 113.06, 8.7) mm, rotated rx 180 ry 0 rz -180 deg; joints [0, 0, 0, 0, 0, 0]
  Call Extruder 0.34896
  MoveL (T6808) to (111.94, 121.16, 8.7) mm, rotated rx 180 ry 0 rz -180 deg; joints [0, 0, 0, 0, 0, 0]
  Call Extruder 0.03385
  MoveL (T6809) to (113.06, 121.16, 8.7) mm, rotated rx 180 ry 0 rz -180 deg; joints [0, 0, 0, 0, 0, 0]
  Call Extruder 0.29531
  MoveL (T6810) to (119.91, 114.3, 8.7) mm, rotated rx 180 ry 0 rz -180 deg; joints [0, 0, 0, 0, 0, 0]
  Call Extruder 0.03794
  MoveL (T6811) to (121.16, 114.3, 8.7) mm, rotated rx 180 ry 0 rz -180 deg; joints [0, 0, 0, 0, 0, 0]
  Call Extruder 0.03647
  MoveL (T6812) to (121.16, 115.5, 8.7) mm, rotated rx 180 ry 0 rz -180 deg; joints [0, 0, 0, 0, 0, 0]
  Set speed (45.0 mm/s)
  Call Extruder -1.6
  MoveL (T6813) to (121.16, 115.5, 8.7) mm, rotated rx 180 ry 0 rz -180 deg; joints [0, 0, 0, 0, 0, 0]
  Set speed (120.0 mm/s)
  MoveL (T6814) to (121.16, 115.5, 8.7) mm, rotated rx 180 ry 0 rz -180 deg; joints [0, 0, 0, 0, 0, 0]
  Call Extruder -0.38
  MoveL (T6815) to (121.16, 114.43, 8.7) mm, rotated rx 180 ry 0 rz -180 deg; joints [0, 0, 0, 0, 0, 0]
  Set speed (45.0 mm/s)
  Call Extruder -0.02
  MoveL (T6816) to (121.16, 114.43, 8.7) mm, rotated rx 180 ry 0 rz -180 deg; joints [0, 0, 0, 0, 0, 0]
  Set speed (150.0 mm/s)
  MoveL (T6817) to (121.16, 114.43, 10.7) mm, rotated rx 180 ry 0 rz -180 deg; joints [0, 0, 0, 0, 0, 0]
  MoveL (T6818) to (104.34, 103.54, 10.7) mm, rotated rx 180 ry 0 rz -180 deg; joints [0, 0, 0, 0, 0, 0]
  MoveL (T6819) to (104.34, 103.54, 8.9) mm, rotated rx 180 ry 0 rz -180 deg; joints [0, 0, 0, 0, 0, 0]
  Set speed (40.0 mm/s)
  Call Extruder 2.0
  MoveL (T6820) to (104.34, 103.54, 8.9) mm, rotated rx 180 ry 0 rz -180 deg; joints [0, 0, 0, 0, 0, 0]
  Set speed (24.9 mm/s)
  MoveL (T6821) to (104.34, 103.54, 8.9) mm, rotated rx 180 ry 0 rz -180 deg; joints [0, 0, 0, 0, 0, 0]
  Call Extruder 0.15245
  MoveL (T6822) to (109.34, 103.54, 8.9) mm, rotated rx 180 ry 0 rz -180 deg; joints [0, 0, 0, 0, 0, 0]
  Call Extruder 0.05775
  MoveL (T6823) to (109.34, 105.44, 8.9) mm, rotated rx 180 ry 0 rz -180 deg; joints [0, 0, 0, 0, 0, 0]
  Call Extruder 0.16065
  MoveL (T6824) to (114.62, 105.44, 8.9) mm, rotated rx 180 ry 0 rz -180 deg; joints [0, 0, 0, 0, 0, 0]
  Call Extruder 0.05775
  MoveL (T6825) to (114.62, 103.54, 8.9) mm, rotated rx 180 ry 0 rz -180 deg; joints [0, 0, 0, 0, 0, 0]
  Call Extruder 0.20844
  MoveL (T6826) to (121.46, 103.54, 8.9) mm, rotated rx 180 ry 0 rz -180 deg; joints [0, 0, 0, 0, 0, 0]
  Call Extruder 0.20399
  MoveL (T6827) to (121.46, 110.23, 8.9) mm, rotated rx 180 ry 0 rz -180 deg; joints [0, 0, 0, 0, 0, 0]
  Call Extruder 0.05901
  MoveL (T6828) to (119.52, 110.23, 8.9) mm, rotated rx 180 ry 0 rz -180 deg; joints [0, 0, 0, 0, 0, 0]
  Call Extruder 0.11452
  MoveL (T6829) to (119.52, 113.99, 8.9) mm, rotated rx 180 ry 0 rz -180 deg; joints [0, 0, 0, 0, 0, 0]
  Call Extruder 0.05906
  MoveL (T6830) to (121.46, 113.99, 8.9) mm, rotated rx 180 ry 0 rz -180 deg; joints [0, 0, 0, 0, 0, 0]
  Call Extruder 0.22746
  MoveL (T6831) to (121.46, 121.46, 8.9) mm, rotated rx 180 ry 0 rz -180 deg; joints [0, 0, 0, 0, 0, 0]
  Call Extruder 0.54596
  MoveL (T6832) to (103.54, 121.46, 8.9) mm, rotated rx 180 ry 0 rz -180 deg; joints [0, 0, 0, 0, 0, 0]
  Call Extruder 0.54596
  MoveL (T6833) to (103.54, 103.54, 8.9) mm, rotated rx 180 ry 0 rz -180 deg; joints [0, 0, 0, 0, 0, 0]
  Call Extruder 0.02254
  MoveL (T6834) to (104.28, 103.54, 8.9) mm, rotated rx 180 ry 0 rz -180 deg; joints [0, 0, 0, 0, 0, 0]
  Set speed (150.0 mm/s)
  MoveL (T6835) to (103.53, 103.13, 8.9) mm, rotated rx 180 ry 0 rz -180 deg; joints [0, 0, 0, 0, 0, 0]
  Set speed (24.9 mm/s)
  MoveL (T6836) to (103.53, 103.13, 8.9) mm, rotated rx 180 ry 0 rz -180 deg; joints [0, 0, 0, 0, 0, 0]
  Call Extruder 0.18943
  MoveL (T6837) to (109.75, 103.13, 8.9) mm, rotated rx 180 ry 0 rz -180 deg; joints [0, 0, 0, 0, 0, 0]
  Call Extruder 0.05775
  MoveL (T6838) to (109.75, 105.03, 8.9) mm, rotated rx 180 ry 0 rz -180 deg; joints [0, 0, 0, 0, 0, 0]
  Call Extruder 0.13586
  MoveL (T6839) to (114.21, 105.03, 8.9) mm, rotated rx 180 ry 0 rz -180 deg; joints [0, 0, 0, 0, 0, 0]
  Call Extruder 0.05775
  MoveL (T6840) to (114.21, 103.13, 8.9) mm, rotated rx 180 ry 0 rz -180 deg; joints [0, 0, 0, 0, 0, 0]
  Call Extruder 0.23324
  MoveL (T6841) to (121.87, 103.13, 8.9) mm, rotated rx 180 ry 0 rz -180 deg; joints [0, 0, 0, 0, 0, 0]
  Call Extruder 0.22879
  MoveL (T6842) to (121.87, 110.64, 8.9) mm, rotated rx 180 ry 0 rz -180 deg; joints [0, 0, 0, 0, 0, 0]
  Call Extruder 0.05902
  MoveL (T6843) to (119.93, 110.64, 8.9) mm, rotated rx 180 ry 0 rz -180 deg; joints [0, 0, 0, 0, 0, 0]
  Call Extruder 0.08971
  MoveL (T6844) to (119.93, 113.59, 8.9) mm, rotated rx 180 ry 0 rz -180 deg; joints [0, 0, 0, 0, 0, 0]
  Call Extruder 0.05906
  MoveL (T6845) to (121.87, 113.59, 8.9) mm, rotated rx 180 ry 0 rz -180 deg; joints [0, 0, 0, 0, 0, 0]
  Call Extruder 0.25226
  MoveL (T6846) to (121.87, 121.87, 8.9) mm, rotated rx 180 ry 0 rz -180 deg; joints [0, 0, 0, 0, 0, 0]
  Call Extruder 0.57077
  MoveL (T6847) to (103.13, 121.87, 8.9) mm, rotated rx 180 ry 0 rz -180 deg; joints [0, 0, 0, 0, 0, 0]
  Call Extruder 0.57077
  MoveL (T6848) to (103.13, 103.13, 8.9) mm, rotated rx 180 ry 0 rz -180 deg; joints [0, 0, 0, 0, 0, 0]
  Call Extruder 0.01036
  MoveL (T6849) to (103.47, 103.13, 8.9) mm, rotated rx 180 ry 0 rz -180 deg; joints [0, 0, 0, 0, 0, 0]
  Set speed (150.0 mm/s)
  MoveL (T6850) to (102.72, 102.81, 8.9) mm, rotated rx 180 ry 0 rz -180 deg; joints [0, 0, 0, 0, 0, 0]
  Set speed (24.9 mm/s)
  MoveL (T6851) to (102.72, 102.81, 8.9) mm, rotated rx 180 ry 0 rz -180 deg; joints [0, 0, 0, 0, 0, 0]
  Call Extruder 0.00259
  MoveL (T6852) to (102.72, 102.72, 8.9) mm, rotated rx 180 ry 0 rz -180 deg; joints [0, 0, 0, 0, 0, 0]
  Call Extruder 0.22641
  MoveL (T6853) to (110.16, 102.72, 8.9) mm, rotated rx 180 ry 0 rz -180 deg; joints [0, 0, 0, 0, 0, 0]
  Call Extruder 0.05775
  MoveL (T6854) to (110.16, 104.62, 8.9) mm, rotated rx 180 ry 0 rz -180 deg; joints [0, 0, 0, 0, 0, 0]
  Call Extruder 0.11107
  MoveL (T6855) to (113.8, 104.62, 8.9) mm, rotated rx 180 ry 0 rz -180 deg; joints [0, 0, 0, 0, 0, 0]
  Call Extruder 0.05775
  MoveL (T6856) to (113.81, 102.72, 8.9) mm, rotated rx 180 ry 0 rz -180 deg; joints [0, 0, 0, 0, 0, 0]
  Call Extruder 0.25803
  MoveL (T6857) to (122.28, 102.72, 8.9) mm, rotated rx 180 ry 0 rz -180 deg; joints [0, 0, 0, 0, 0, 0]
  Call Extruder 0.2536
  MoveL (T6858) to (122.28, 111.05, 8.9) mm, rotated rx 180 ry 0 rz -180 deg; joints [0, 0, 0, 0, 0, 0]
  Call Extruder 0.05902
  MoveL (T6859) to (120.34, 111.05, 8.9) mm, rotated rx 180 ry 0 rz -180 deg; joints [0, 0, 0, 0, 0, 0]
  Call Extruder 0.06491
  MoveL (T6860) to (120.34, 113.18, 8.9) mm, rotated rx 180 ry 0 rz -180 deg; joints [0, 0, 0, 0, 0, 0]
  Call Extruder 0.05905
  MoveL (T6861) to (122.28, 113.18, 8.9) mm, rotated rx 180 ry 0 rz -180 deg; joints [0, 0, 0, 0, 0, 0]
  Call Extruder 0.27706
  MoveL (T6862) to (122.28, 122.28, 8.9) mm, rotated rx 180 ry 0 rz -180 deg; joints [0, 0, 0, 0, 0, 0]
  Call Extruder 0.59557
  MoveL (T6863) to (102.72, 122.28, 8.9) mm, rotated rx 180 ry 0 rz -180 deg; joints [0, 0, 0, 0, 0, 0]
  Call Extruder 0.59115
  MoveL (T6864) to (102.72, 102.87, 8.9) mm, rotated rx 180 ry 0 rz -180 deg; joints [0, 0, 0, 0, 0, 0]
  Set speed (150.0 mm/s)
  MoveL (T6865) to (102.78, 102.75, 8.9) mm, rotated rx 180 ry 0 rz -180 deg; joints [0, 0, 0, 0, 0, 0]
  Set speed (45.0 mm/s)
  Call Extruder -1.6
  MoveL (T6866) to (102.78, 102.75, 8.9) mm, rotated rx 180 ry 0 rz -180 deg; joints [0, 0, 0, 0, 0, 0]
  Set speed (120.0 mm/s)
  MoveL (T6867) to (102.78, 102.75, 8.9) mm, rotated rx 180 ry 0 rz -180 deg; joints [0, 0, 0, 0, 0, 0]
  Call Extruder -0.05166
  MoveL (T6868) to (102.72, 102.72, 8.9) mm, rotated rx 180 ry 0 rz -180 deg; joints [0, 0, 0, 0, 0, 0]
  Call Extruder -0.32834
  MoveL (T6869) to (103.65, 102.72, 8.9) mm, rotated rx 180 ry 0 rz -180 deg; joints [0, 0, 0, 0, 0, 0]
  Set speed (45.0 mm/s)
  Call Extruder -0.02
  MoveL (T6870) to (103.65, 102.72, 8.9) mm, rotated rx 180 ry 0 rz -180 deg; joints [0, 0, 0, 0, 0, 0]
  Set speed (150.0 mm/s)
  MoveL (T6871) to (103.65, 102.72, 10.9) mm, rotated rx 180 ry 0 rz -180 deg; joints [0, 0, 0, 0, 0, 0]
  MoveL (T6872) to (106.29, 103.84, 10.9) mm, rotated rx 180 ry 0 rz -180 deg; joints [0, 0, 0, 0, 0, 0]
  MoveL (T6873) to (106.29, 103.84, 8.9) mm, rotated rx 180 ry 0 rz -180 deg; joints [0, 0, 0, 0, 0, 0]
  Set speed (40.0 mm/s)
  Call Extruder 2.0
  MoveL (T6874) to (106.29, 103.84, 8.9) mm, rotated rx 180 ry 0 rz -180 deg; joints [0, 0, 0, 0, 0, 0]
  Set speed (24.9 mm/s)
  MoveL (T6875) to (106.29, 103.84, 8.9) mm, rotated rx 180 ry 0 rz -180 deg; joints [0, 0, 0, 0, 0, 0]
  Call Extruder 0.07441
  MoveL (T6876) to (103.84, 103.84, 8.9) mm, rotated rx 180 ry 0 rz -180 deg; joints [0, 0, 0, 0, 0, 0]
  Call Extruder 0.7458
  MoveL (T6877) to (121.16, 121.16, 8.9) mm, rotated rx 180 ry 0 rz -180 deg; joints [0, 0, 0, 0, 0, 0]
  Call Extruder 0.07441
  MoveL (T6878) to (118.71, 121.16, 8.9) mm, rotated rx 180 ry 0 rz -180 deg; joints [0, 0, 0, 0, 0, 0]
  Set speed (45.0 mm/s)
  Call Extruder -1.6
  MoveL (T6879) to (118.71, 121.16, 8.9) mm, rotated rx 180 ry 0 rz -180 deg; joints [0, 0, 0, 0, 0, 0]
  Set speed (120.0 mm/s)
  MoveL (T6880) to (118.71, 121.16, 8.9) mm, rotated rx 180 ry 0 rz -180 deg; joints [0, 0, 0, 0, 0, 0]
  Call Extruder -0.38
  MoveL (T6881) to (119.78, 121.16, 8.9) mm, rotated rx 180 ry 0 rz -180 deg; joints [0, 0, 0, 0, 0, 0]
  Set speed (45.0 mm/s)
  Call Extruder -0.02
  MoveL (T6882) to (119.78, 121.16, 8.9) mm, rotated rx 180 ry 0 rz -180 deg; joints [0, 0, 0, 0, 0, 0]
  Set speed (150.0 mm/s)
  MoveL (T6883) to (119.78, 121.16, 10.9) mm, rotated rx 180 ry 0 rz -180 deg; joints [0, 0, 0, 0, 0, 0]
  MoveL (T6884) to (120.89, 114.12, 10.9) mm, rotated rx 180 ry 0 rz -180 deg; joints [0, 0, 0, 0, 0, 0]
  MoveL (T6885) to (120.89, 114.12, 8.9) mm, rotated rx 180 ry 0 rz -180 deg; joints [0, 0, 0, 0, 0, 0]
  Set speed (40.0 mm/s)
  Call Extruder 2.0
  MoveL (T6886) to (120.89, 114.12, 8.9) mm, rotated rx 180 ry 0 rz -180 deg; joints [0, 0, 0, 0, 0, 0]
  Set speed (24.9 mm/s)
  MoveL (T6887) to (120.89, 114.12, 8.9) mm, rotated rx 180 ry 0 rz -180 deg; joints [0, 0, 0, 0, 0, 0]
  Call Extruder 0.01551
  MoveL (T6888) to (120.56, 114.45, 8.9) mm, rotated rx 180 ry 0 rz -180 deg; joints [0, 0, 0, 0, 0, 0]
  Call Extruder 0.02033
  MoveL (T6889) to (119.94, 114.45, 8.9) mm, rotated rx 180 ry 0 rz -180 deg; joints [0, 0, 0, 0, 0, 0]
  Call Extruder 0.01549
  MoveL (T6890) to (120.28, 114.12, 8.9) mm, rotated rx 180 ry 0 rz -180 deg; joints [0, 0, 0, 0, 0, 0]
  Set speed (45.0 mm/s)
  Call Extruder -1.6
  MoveL (T6891) to (120.28, 114.12, 8.9) mm, rotated rx 180 ry 0 rz -180 deg; joints [0, 0, 0, 0, 0, 0]
  Set speed (120.0 mm/s)
  MoveL (T6892) to (120.28, 114.12, 8.9) mm, rotated rx 180 ry 0 rz -180 deg; joints [0, 0, 0, 0, 0, 0]
  Call Extruder -0.1681
  MoveL (T6893) to (119.94, 114.45, 8.9) mm, rotated rx 180 ry 0 rz -180 deg; joints [0, 0, 0, 0, 0, 0]
  Call Extruder -0.2119
  MoveL (T6894) to (120.54, 114.45, 8.9) mm, rotated rx 180 ry 0 rz -180 deg; joints [0, 0, 0, 0, 0, 0]
  Set speed (45.0 mm/s)
  Call Extruder -0.02
  MoveL (T6895) to (120.54, 114.45, 8.9) mm, rotated rx 180 ry 0 rz -180 deg; joints [0, 0, 0, 0, 0, 0]
  Set speed (150.0 mm/s)
  MoveL (T6896) to (120.54, 114.45, 10.9) mm, rotated rx 180 ry 0 rz -180 deg; joints [0, 0, 0, 0, 0, 0]
  MoveL (T6897) to (119.22, 112.09, 10.9) mm, rotated rx 180 ry 0 rz -180 deg; joints [0, 0, 0, 0, 0, 0]
  MoveL (T6898) to (119.22, 112.09, 8.9) mm, rotated rx 180 ry 0 rz -180 deg; joints [0, 0, 0, 0, 0, 0]
  Set speed (40.0 mm/s)
  Call Extruder 2.0
  MoveL (T6899) to (119.22, 112.09, 8.9) mm, rotated rx 180 ry 0 rz -180 deg; joints [0, 0, 0, 0, 0, 0]
  Set speed (24.9 mm/s)
  MoveL (T6900) to (119.22, 112.09, 8.9) mm, rotated rx 180 ry 0 rz -180 deg; joints [0, 0, 0, 0, 0, 0]
  Call Extruder 0.0567
  MoveL (T6901) to (119.22, 113.96, 8.9) mm, rotated rx 180 ry 0 rz -180 deg; joints [0, 0, 0, 0, 0, 0]
  Call Extruder 0.00549
  MoveL (T6902) to (119.09, 114.08, 8.9) mm, rotated rx 180 ry 0 rz -180 deg; joints [0, 0, 0, 0, 0, 0]
  Call Extruder 0.01221
  MoveL (T6903) to (119.09, 114.48, 8.9) mm, rotated rx 180 ry 0 rz -180 deg; joints [0, 0, 0, 0, 0, 0]
  Call Extruder 0.37674
  MoveL (T6904) to (110.35, 105.74, 8.9) mm, rotated rx 180 ry 0 rz -180 deg; joints [0, 0, 0, 0, 0, 0]
  Call Extruder 0.00904
  MoveL (T6905) to (110.05, 105.74, 8.9) mm, rotated rx 180 ry 0 rz -180 deg; joints [0, 0, 0, 0, 0, 0]
  Call Extruder 0.2673
  MoveL (T6906) to (103.84, 111.94, 8.9) mm, rotated rx 180 ry 0 rz -180 deg; joints [0, 0, 0, 0, 0, 0]
  Call Extruder 0.03385
  MoveL (T6907) to (103.84, 113.06, 8.9) mm, rotated rx 180 ry 0 rz -180 deg; joints [0, 0, 0, 0, 0, 0]
  Call Extruder 0.34896
  MoveL (T6908) to (111.94, 121.16, 8.9) mm, rotated rx 180 ry 0 rz -180 deg; joints [0, 0, 0, 0, 0, 0]
  Call Extruder 0.03385
  MoveL (T6909) to (113.06, 121.16, 8.9) mm, rotated rx 180 ry 0 rz -180 deg; joints [0, 0, 0, 0, 0, 0]
  Call Extruder 0.27257
  MoveL (T6910) to (119.38, 114.83, 8.9) mm, rotated rx 180 ry 0 rz -180 deg; joints [0, 0, 0, 0, 0, 0]
  Call Extruder 0.00117
  MoveL (T6911) to (119.41, 114.86, 8.9) mm, rotated rx 180 ry 0 rz -180 deg; joints [0, 0, 0, 0, 0, 0]
  Call Extruder 0.00159
  MoveL (T6912) to (119.46, 114.86, 8.9) mm, rotated rx 180 ry 0 rz -180 deg; joints [0, 0, 0, 0, 0, 0]
  Call Extruder 0.07298
  MoveL (T6913) to (121.16, 116.55, 8.9) mm, rotated rx 180 ry 0 rz -180 deg; joints [0, 0, 0, 0, 0, 0]
  Call Extruder 0.03385
  MoveL (T6914) to (121.16, 117.66, 8.9) mm, rotated rx 180 ry 0 rz -180 deg; joints [0, 0, 0, 0, 0, 0]
  Call Extruder 0.15054
  MoveL (T6915) to (117.66, 121.16, 8.9) mm, rotated rx 180 ry 0 rz -180 deg; joints [0, 0, 0, 0, 0, 0]
  Call Extruder 0.03385
  MoveL (T6916) to (116.55, 121.16, 8.9) mm, rotated rx 180 ry 0 rz -180 deg; joints [0, 0, 0, 0, 0, 0]
  Call Extruder 0.54738
  MoveL (T6917) to (103.84, 108.45, 8.9) mm, rotated rx 180 ry 0 rz -180 deg; joints [0, 0, 0, 0, 0, 0]
  Call Extruder 0.03385
  MoveL (T6918) to (103.84, 107.34, 8.9) mm, rotated rx 180 ry 0 rz -180 deg; joints [0, 0, 0, 0, 0, 0]
  Call Extruder 0.15054
  MoveL (T6919) to (107.34, 103.84, 8.9) mm, rotated rx 180 ry 0 rz -180 deg; joints [0, 0, 0, 0, 0, 0]
  Call Extruder 0.03385
  MoveL (T6920) to (108.45, 103.84, 8.9) mm, rotated rx 180 ry 0 rz -180 deg; joints [0, 0, 0, 0, 0, 0]
  Call Extruder 0.00068
  MoveL (T6921) to (108.47, 103.86, 8.9) mm, rotated rx 180 ry 0 rz -180 deg; joints [0, 0, 0, 0, 0, 0]
  Call Extruder 0.05143
  MoveL (T6922) to (108.47, 105.55, 8.9) mm, rotated rx 180 ry 0 rz -180 deg; joints [0, 0, 0, 0, 0, 0]
  Call Extruder 0.01375
  MoveL (T6923) to (108.79, 105.87, 8.9) mm, rotated rx 180 ry 0 rz -180 deg; joints [0, 0, 0, 0, 0, 0]
  Call Extruder 0.00923
  MoveL (T6924) to (109.09, 105.87, 8.9) mm, rotated rx 180 ry 0 rz -180 deg; joints [0, 0, 0, 0, 0, 0]
  Set speed (150.0 mm/s)
  MoveL (T6925) to (109.22, 104.69, 8.9) mm, rotated rx 180 ry 0 rz -180 deg; joints [0, 0, 0, 0, 0, 0]
  Set speed (24.9 mm/s)
  MoveL (T6926) to (109.22, 104.69, 8.9) mm, rotated rx 180 ry 0 rz -180 deg; joints [0, 0, 0, 0, 0, 0]
  Call Extruder 0.01598
  MoveL (T6927) to (108.87, 105.04, 8.9) mm, rotated rx 180 ry 0 rz -180 deg; joints [0, 0, 0, 0, 0, 0]
  Call Extruder 0.01988
  MoveL (T6928) to (108.87, 104.43, 8.9) mm, rotated rx 180 ry 0 rz -180 deg; joints [0, 0, 0, 0, 0, 0]
  Call Extruder 0.01598
  MoveL (T6929) to (109.22, 104.08, 8.9) mm, rotated rx 180 ry 0 rz -180 deg; joints [0, 0, 0, 0, 0, 0]
  Set speed (45.0 mm/s)
  Call Extruder -1.6
  MoveL (T6930) to (109.22, 104.08, 8.9) mm, rotated rx 180 ry 0 rz -180 deg; joints [0, 0, 0, 0, 0, 0]
  Set speed (120.0 mm/s)
  MoveL (T6931) to (109.22, 104.08, 8.9) mm, rotated rx 180 ry 0 rz -180 deg; joints [0, 0, 0, 0, 0, 0]
  Call Extruder -0.17547
  MoveL (T6932) to (108.87, 104.43, 8.9) mm, rotated rx 180 ry 0 rz -180 deg; joints [0, 0, 0, 0, 0, 0]
  Call Extruder -0.20453
  MoveL (T6933) to (108.87, 105, 8.9) mm, rotated rx 180 ry 0 rz -180 deg; joints [0, 0, 0, 0, 0, 0]
  Set speed (45.0 mm/s)
  Call Extruder -0.02
  MoveL (T6934) to (108.87, 105, 8.9) mm, rotated rx 180 ry 0 rz -180 deg; joints [0, 0, 0, 0, 0, 0]
  Set speed (150.0 mm/s)
  MoveL (T6935) to (108.87, 105, 10.9) mm, rotated rx 180 ry 0 rz -180 deg; joints [0, 0, 0, 0, 0, 0]
  MoveL (T6936) to (114.87, 105.64, 10.9) mm, rotated rx 180 ry 0 rz -180 deg; joints [0, 0, 0, 0, 0, 0]
  MoveL (T6937) to (114.87, 105.64, 8.9) mm, rotated rx 180 ry 0 rz -180 deg; joints [0, 0, 0, 0, 0, 0]
  Set speed (40.0 mm/s)
  Call Extruder 2.0
  MoveL (T6938) to (114.87, 105.64, 8.9) mm, rotated rx 180 ry 0 rz -180 deg; joints [0, 0, 0, 0, 0, 0]
  Set speed (24.9 mm/s)
  MoveL (T6939) to (114.87, 105.64, 8.9) mm, rotated rx 180 ry 0 rz -180 deg; joints [0, 0, 0, 0, 0, 0]
  Call Extruder 0.01303
  MoveL (T6940) to (115.15, 105.36, 8.9) mm, rotated rx 180 ry 0 rz -180 deg; joints [0, 0, 0, 0, 0, 0]
  Call Extruder 0.01996
  MoveL (T6941) to (115.15, 104.75, 8.9) mm, rotated rx 180 ry 0 rz -180 deg; joints [0, 0, 0, 0, 0, 0]
  Call Extruder 0.01044
  MoveL (T6942) to (114.92, 104.97, 8.9) mm, rotated rx 180 ry 0 rz -180 deg; joints [0, 0, 0, 0, 0, 0]
  Call Extruder 0.01996
  MoveL (T6943) to (114.92, 104.36, 8.9) mm, rotated rx 180 ry 0 rz -180 deg; joints [0, 0, 0, 0, 0, 0]
  Call Extruder 0.01886
  MoveL (T6944) to (115.33, 103.95, 8.9) mm, rotated rx 180 ry 0 rz -180 deg; joints [0, 0, 0, 0, 0, 0]
  Set speed (150.0 mm/s)
  MoveL (T6945) to (116.35, 103.84, 8.9) mm, rotated rx 180 ry 0 rz -180 deg; joints [0, 0, 0, 0, 0, 0]
  Set speed (24.9 mm/s)
  MoveL (T6946) to (116.35, 103.84, 8.9) mm, rotated rx 180 ry 0 rz -180 deg; joints [0, 0, 0, 0, 0, 0]
  Call Extruder 0.02402
  MoveL (T6947) to (115.56, 103.84, 8.9) mm, rotated rx 180 ry 0 rz -180 deg; joints [0, 0, 0, 0, 0, 0]
  Call Extruder 0.03024
  MoveL (T6948) to (115.56, 104.84, 8.9) mm, rotated rx 180 ry 0 rz -180 deg; joints [0, 0, 0, 0, 0, 0]
  Call Extruder 0.04276
  MoveL (T6949) to (116.55, 103.84, 8.9) mm, rotated rx 180 ry 0 rz -180 deg; joints [0, 0, 0, 0, 0, 0]
  Call Extruder 0.03385
  MoveL (T6950) to (117.66, 103.84, 8.9) mm, rotated rx 180 ry 0 rz -180 deg; joints [0, 0, 0, 0, 0, 0]
  Call Extruder 0.15054
  MoveL (T6951) to (121.16, 107.34, 8.9) mm, rotated rx 180 ry 0 rz -180 deg; joints [0, 0, 0, 0, 0, 0]
  Call Extruder 0.03385
  MoveL (T6952) to (121.16, 108.45, 8.9) mm, rotated rx 180 ry 0 rz -180 deg; joints [0, 0, 0, 0, 0, 0]
  Call Extruder 0.03779
  MoveL (T6953) to (120.28, 109.33, 8.9) mm, rotated rx 180 ry 0 rz -180 deg; joints [0, 0, 0, 0, 0, 0]
  Call Extruder 0.02672
  MoveL (T6954) to (121.16, 109.33, 8.9) mm, rotated rx 180 ry 0 rz -180 deg; joints [0, 0, 0, 0, 0, 0]
  Call Extruder 0.02051
  MoveL (T6955) to (121.16, 108.65, 8.9) mm, rotated rx 180 ry 0 rz -180 deg; joints [0, 0, 0, 0, 0, 0]
  Set speed (150.0 mm/s)
  MoveL (T6956) to (121.02, 109.55, 8.9) mm, rotated rx 180 ry 0 rz -180 deg; joints [0, 0, 0, 0, 0, 0]
  Set speed (24.9 mm/s)
  MoveL (T6957) to (121.02, 109.55, 8.9) mm, rotated rx 180 ry 0 rz -180 deg; joints [0, 0, 0, 0, 0, 0]
  Call Extruder 0.01748
  MoveL (T6958) to (120.64, 109.93, 8.9) mm, rotated rx 180 ry 0 rz -180 deg; joints [0, 0, 0, 0, 0, 0]
  Call Extruder 0.02011
  MoveL (T6959) to (120.02, 109.93, 8.9) mm, rotated rx 180 ry 0 rz -180 deg; joints [0, 0, 0, 0, 0, 0]
  Call Extruder 0.009
  MoveL (T6960) to (120.22, 109.73, 8.9) mm, rotated rx 180 ry 0 rz -180 deg; joints [0, 0, 0, 0, 0, 0]
  Call Extruder 0.02013
  MoveL (T6961) to (119.6, 109.73, 8.9) mm, rotated rx 180 ry 0 rz -180 deg; joints [0, 0, 0, 0, 0, 0]
  Call Extruder 0.01314
  MoveL (T6962) to (119.31, 110.02, 8.9) mm, rotated rx 180 ry 0 rz -180 deg; joints [0, 0, 0, 0, 0, 0]
  Set speed (45.0 mm/s)
  Call Extruder -1.6
  MoveL (T6963) to (119.31, 110.02, 8.9) mm, rotated rx 180 ry 0 rz -180 deg; joints [0, 0, 0, 0, 0, 0]
  Set speed (120.0 mm/s)
  MoveL (T6964) to (119.31, 110.02, 8.9) mm, rotated rx 180 ry 0 rz -180 deg; joints [0, 0, 0, 0, 0, 0]
  Call Extruder -0.14349
  MoveL (T6965) to (119.6, 109.73, 8.9) mm, rotated rx 180 ry 0 rz -180 deg; joints [0, 0, 0, 0, 0, 0]
  Call Extruder -0.21975
  MoveL (T6966) to (120.22, 109.73, 8.9) mm, rotated rx 180 ry 0 rz -180 deg; joints [0, 0, 0, 0, 0, 0]
  Call Extruder -0.01676
  MoveL (T6967) to (120.18, 109.77, 8.9) mm, rotated rx 180 ry 0 rz -180 deg; joints [0, 0, 0, 0, 0, 0]
  Set speed (45.0 mm/s)
  Call Extruder -0.02
  MoveL (T6968) to (120.18, 109.77, 8.9) mm, rotated rx 180 ry 0 rz -180 deg; joints [0, 0, 0, 0, 0, 0]
  Set speed (150.0 mm/s)
  MoveL (T6969) to (120.18, 109.77, 10.9) mm, rotated rx 180 ry 0 rz -180 deg; joints [0, 0, 0, 0, 0, 0]
  MoveL (T6970) to (118.71, 103.84, 10.9) mm, rotated rx 180 ry 0 rz -180 deg; joints [0, 0, 0, 0, 0, 0]
  MoveL (T6971) to (118.71, 103.84, 8.9) mm, rotated rx 180 ry 0 rz -180 deg; joints [0, 0, 0, 0, 0, 0]
  Set speed (40.0 mm/s)
  Call Extruder 2.0
  MoveL (T6972) to (118.71, 103.84, 8.9) mm, rotated rx 180 ry 0 rz -180 deg; joints [0, 0, 0, 0, 0, 0]
  Set speed (24.9 mm/s)
  MoveL (T6973) to (118.71, 103.84, 8.9) mm, rotated rx 180 ry 0 rz -180 deg; joints [0, 0, 0, 0, 0, 0]
  Call Extruder 0.07441
  MoveL (T6974) to (121.16, 103.84, 8.9) mm, rotated rx 180 ry 0 rz -180 deg; joints [0, 0, 0, 0, 0, 0]
  Call Extruder 0.7458
  MoveL (T6975) to (103.84, 121.16, 8.9) mm, rotated rx 180 ry 0 rz -180 deg; joints [0, 0, 0, 0, 0, 0]
  Call Extruder 0.10645
  MoveL (T6976) to (103.84, 117.66, 8.9) mm, rotated rx 180 ry 0 rz -180 deg; joints [0, 0, 0, 0, 0, 0]
  Call Extruder 0.15054
  MoveL (T6977) to (107.34, 121.16, 8.9) mm, rotated rx 180 ry 0 rz -180 deg; joints [0, 0, 0, 0, 0, 0]
  Call Extruder 0.03385
  MoveL (T6978) to (108.45, 121.16, 8.9) mm, rotated rx 180 ry 0 rz -180 deg; joints [0, 0, 0, 0, 0, 0]
  Call Extruder 0.46392
  MoveL (T6979) to (119.22, 110.39, 8.9) mm, rotated rx 180 ry 0 rz -180 deg; joints [0, 0, 0, 0, 0, 0]
  Call Extruder 0.00352
  MoveL (T6980) to (119.22, 110.27, 8.9) mm, rotated rx 180 ry 0 rz -180 deg; joints [0, 0, 0, 0, 0, 0]
  Call Extruder 0.00551
  MoveL (T6981) to (119.09, 110.14, 8.9) mm, rotated rx 180 ry 0 rz -180 deg; joints [0, 0, 0, 0, 0, 0]
  Call Extruder 0.00802
  MoveL (T6982) to (119.09, 109.88, 8.9) mm, rotated rx 180 ry 0 rz -180 deg; joints [0, 0, 0, 0, 0, 0]
  Call Extruder 0.17288
  MoveL (T6983) to (115.08, 105.87, 8.9) mm, rotated rx 180 ry 0 rz -180 deg; joints [0, 0, 0, 0, 0, 0]
  Call Extruder 0.01131
  MoveL (T6984) to (114.71, 105.87, 8.9) mm, rotated rx 180 ry 0 rz -180 deg; joints [0, 0, 0, 0, 0, 0]
  Call Extruder 0.00391
  MoveL (T6985) to (114.62, 105.78, 8.9) mm, rotated rx 180 ry 0 rz -180 deg; joints [0, 0, 0, 0, 0, 0]
